         //Temporärer Fehler: #pdStatus = 80A7, 80B5, 80C0, 80C1, 80C2, 80C3 oder 80C4 zulassen und nocheinmal versuchen
         IF NOT (#pwWord1 = DW#16#80A7) AND NOT (#pwWord1 = DW#16#80B5) AND NOT (#pwWord1 = DW#16#80C0) AND
           NOT (#pwWord1 = DW#16#80C1) AND NOT (#pwWord1 = DW#16#80C2) AND NOT (#pwWord1 = DW#16#80C3) AND
           NOT (#pwWord1 = DW#16#80C4) THEN

           // Wiederholungsauftrag wieder zurücknehmen
           #sbWrStart2 := False;
           #sbRdStart2 := False;
           #sbWrite := False;

           // Fehler ausgeben 
           #sbError := #sbRdError;

         ELSE
           // Fehlerwiederholauftrag ??                   
           IF #siErrorCount = #siMaxErrCount THEN

             // Wiederholungsauftrag wieder zurücknehmen
             #sbWrStart2 := False;
             #sbRdStart2 := False;
             #sbWrite := False;

             //Fehlerzähler zurücksetzen
             #siErrorCount := 0;


             // Fehler ausgeben 
             #sbError := #sbRdError;

             // nix tun bis Zähler überläuft
           ELSE
             #siErrorCount := #siErrorCount + 1;
           END_IF;
         END_IF;

         // Fehler : die Auftragsreferenz der Antwort übertimmt nicht mit der Auftragsreferenz der Anfrage überein
       ELSIF NOT (#siReqRef = BYTE_TO_INT(#sxRespParaMulti.sxHeader.syReqRef)) AND NOT #sbRdBusy AND #pbValidSFB THEN
         #siErrorId := 1;
         #sbError := True;
         #sbDone := False;

         // Wiederholungsauftrag wieder zurücknehmen
         #sbWrStart2 := False;
         #sbRdStart2 := False;
         #sbWrite := False;

         // Fehler : falsche Auftragskennung zurück erhalten    
       ELSIF NOT (#sxRespParaMulti.sxHeader.syReqId = B#16#82 OR #sxRespParaMulti.sxHeader.syReqId = B#16#02) AND
         NOT #sbRdBusy AND #pbValidSFB THEN
         #siErrorId := 1;
         #sbError := True;
         #sbDone := False;

         // Wiederholungsauftrag wieder zurücknehmen
         #sbWrStart2 := False;
         #sbRdStart2 := False;
         #sbWrite := False;

         // Fehler : die angeforderte Anzahl Parameter entspricht nicht der übermittelten Anzahl Parameter überein
       ELSIF NOT (#sxRespParaMulti.sxHeader.syParaNo = B#16#01) AND NOT #sbRdBusy AND #pbValidSFB THEN
         #siErrorId := 1;
         #sbError := True;
         #sbDone := False;

         // Wiederholungsauftrag wieder zurücknehmen
         #sbWrStart2 := False;
         #sbRdStart2 := False;
         #sbWrite := False;

         // Fehler : die Achse entspricht nicht der übergebenen Achse
       ELSIF NOT (#syAxisNo = #sxRespParaMulti.sxHeader.syAxisNo) AND NOT #sbRdBusy AND #pbValidSFB THEN
         #siErrorId := 1;
         #sbError := True;
         #sbDone := False;

         // Wiederholungsauftrag wieder zurücknehmen
         #sbWrStart2 := False;
         #sbRdStart2 := False;
         #sbWrite := False;

         // kein Fehler beim LESEN AZYKLISCH und Auftrag fertig 
       ELSIF NOT #sbRdBusy AND #pbValidSFB THEN

         // 2. Teilauftrag "Parameter schreiben bzw. ändern" negative Rückmeldung erhalten 
         IF #sxRespParaMulti.sxHeader.syReqId = B#16#82 THEN

           // die angefragten Parameter auswerten und im Puffer abspeichern
           // Format des Parameters auswerten, bei Format = Error Fehler auswerten 
           IF (BYTE_TO_INT(#sxRespParaMulti.sxData[1]) = 68) THEN

             // Fehlerwert ermitteln und abspeichern 
             // Format = Word, zwei Bytes zu übermitteltem Parameterwert zusammenfassen
             #pwWordHigh := SHL(IN := BYTE_TO_WORD(#sxRespParaMulti.sxData[3]), N := 8);
             #pwWordLow := BYTE_TO_WORD(#sxRespParaMulti.sxData[4]);
             #pwWord1 := #pwWordHigh XOR #pwWordLow;

             #sbError := True;

             // ermittelte Fehlernummer im Puffer zurücksetzen
             #ErrorNo := W#16#00;

             #ErrorNo := #pwWord1;

             // Die Fehlerhaftigkeit des erkannten Parameter in der Fehlernummer eintragen   
             #swParaError := #swParaError OR W#16#01;

           ELSE

             // Die Fehlerhaftigkeit des erkannten Parameter in der Fehlernummer löschen   
             #swParaError := #swParaError AND W#16#FFFE;

             // ermittelte Fehlernummer im Puffer zurücksetzen
             #ErrorNo := W#16#00;
           END_IF;
         END_IF; // 2. Teilauftrag "Parameter schreiben bzw. ändern" negative Rückmeldung erhalten

         // Fehlerkennung zurücknehmen
         IF (#siErrorId = 3) OR (#siErrorId = 1) THEN
           #siErrorId := 0;
           #sbError := False;
         END_IF;

         #DiagId := W#16#00;

         // 2. Teilauftrag "Parameter schreiben bzw. ändern" ist abgeschlossen
         #sbRdStart2 := False;
         #sbWrite := False;

       END_IF; // kein Fehler beim LESEN AZYKLISCH und Auftrag fertig 
     END_IF; // vom 2. Teilauftrag "Parameter schreiben bzw. ändern" die Antwort abwarten und dann auswerten 
   END_IF; // Auftrag "Parameter schreiben" wurde ausgelöst

   #pdDWordHigh := SHL(IN := INT_TO_DWORD(#siErrorId), N := 16);
   #pdDWordLow := WORD_TO_DWORD(#swParaError);

   // ermittelter Parameterwert eintragen (Word)
   #ErrorId := #pdDWordHigh XOR #pdDWordLow;

   // Initialisierung von Ausgängen
   #Busy := #sbBusy;
   #Error := #sbError;
   #Format := #syFormat;
   // Änderung wegen verhalten von Ready  
   #Done := #sbDone;
   // Prüfen, ob Auftrag abgeschlossen ist
   IF ((#Error OR #Done) AND NOT #sbReady) THEN
     #Ready := True;
     #sbReady := True;
   ELSE
     #Ready := False;
   END_IF;
END_FUNCTION_BLOCK

FUNCTION_BLOCK "SevroStart&PosCheck"   // FB4073, LAD
{ S7_Optimized_Access := 'TRUE' }
// stored: AutoNumber false, MemoryReserve 100, SetENOAutomatically false
   VAR_INPUT
      iRef_Homed { ExternalAccessible := 'False'; ExternalVisible := 'False'; ExternalWritable := 'False'} : Bool;
      iStandstill { ExternalAccessible := 'False'; ExternalVisible := 'False'; ExternalWritable := 'False'} : Bool;
      iReset : Bool;
      interlcok : Bool;   // 启动互锁
      "iActual Posi" { ExternalAccessible := 'False'; ExternalVisible := 'False'; ExternalWritable := 'False'} : DInt;
      "iTol+" { ExternalAccessible := 'False'; ExternalVisible := 'False'; ExternalWritable := 'False'} : DInt;
      "iTol-" { ExternalAccessible := 'False'; ExternalVisible := 'False'; ExternalWritable := 'False'} : DInt;
      iStartTon : Time := T#200ms;   // 启动延迟
   END_VAR
   VAR_OUTPUT
      oStartPos : Bool;   // 启动
      DoublePosError : Bool;   // 多位置触发
   END_VAR
   VAR_IN_OUT
      ioPoint : Array[0..39] of Struct
         Start : Bool;
         Achieve : Bool;
      END_STRUCT;
      ioList : "PosList";
      ioPosNumberSelect : Int;   // 位置启动
   END_VAR
   VAR
      TON : Array[0..1] of TON_TIME;
      StartCount { S7_SetPoint := 'True'} : Int;   // 启动计数
   END_VAR
   VAR_TEMP
      "Actual Posi+Tol" : DInt;
      "Actual Posi-Tol" : DInt;
      Index : Array[0..7] of Int;   // 位置启动
      PosStart : Bool;
   END_VAR
   VAR_TEMP   // added for the SCL form of the ladder/FBD networks
      _w1 : Bool;
   END_VAR
BEGIN

REGION Network 1 (SCL): 检查当前启动位置号
   #Index[1] := 0;
   #PosStart := false;
   FOR #Index[1] := 0 TO 39 DO
       IF #ioPoint[#Index[1]].Start THEN

           #ioPosNumberSelect := #Index[1];//当前启动位置号
           #PosStart := TRUE;
           EXIT;
       END_IF;
   END_FOR;
   #Index[2] := 0;
   #StartCount := 0;
   FOR #Index[2] := 0 TO 39 DO
       IF #ioPoint[#Index[2]].Start THEN

           #StartCount := #StartCount+1;//当前启动位置号


       END_IF;
       IF #Index[2] = 39 THEN

           EXIT;
       END_IF;

   END_FOR;
END_REGION

REGION Network 2: 位置给定
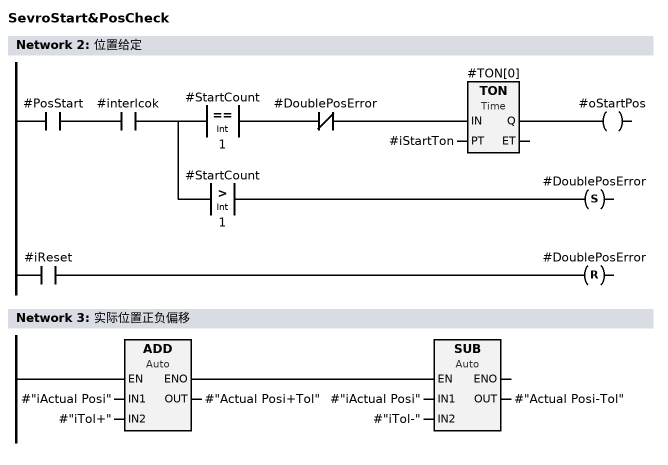
   RUNG wire#powerrail
      Contact( #PosStart )
      Contact( #interlcok )
      wire#w1
      { S7_Templates := "SrcType := Int" } EQ_Contact(in1 := #StartCount, in2 := 1)
      I_Contact( #DoublePosError )
      { S7_Templates := "time_type := Time" } #TON[0].TON(pt := #iStartTon, et =>)
      Coil( #oStartPos )
   END_RUNG
   RUNG wire#w1
      { S7_Templates := "SrcType := Int" } GT_Contact(in1 := #StartCount, in2 := 1)
      S_Coil( #DoublePosError )
   END_RUNG
   RUNG wire#powerrail
      Contact( #iReset )
      R_Coil( #DoublePosError )
   END_RUNG
   // the same network as SCL:
   #_w1 := #PosStart AND #interlcok;
   #TON[0].TON(IN := #_w1 AND (#StartCount = 1) AND NOT #DoublePosError, PT := #iStartTon);
   #oStartPos := #TON[0].Q;
   IF #_w1 AND (#StartCount > 1) THEN #DoublePosError := TRUE; END_IF;
   IF #iReset THEN #DoublePosError := FALSE; END_IF;
END_REGION

REGION Network 3: 实际位置正负偏移
   RUNG wire#powerrail
      Add(in1 := #"iActual Posi", in2 := #"iTol+", out => #"Actual Posi+Tol")
      Sub(in1 := #"iActual Posi", in2 := #"iTol-", out => #"Actual Posi-Tol")
   END_RUNG
   // the same network as SCL:
   #"Actual Posi+Tol" := #"iActual Posi" + #"iTol+";
   #"Actual Posi-Tol" := #"iActual Posi" - #"iTol-";
END_REGION

REGION Network 4 (SCL): 位置检查


   #Index[3] := 0;
   FOR #Index[3] := 0 TO 39 DO
       IF #ioList.List[ #Index[3]].Pos>= #"Actual Posi-Tol"
           AND #ioList.List[ #Index[3]].Pos<= #"Actual Posi+Tol"
       THEN
         #ioPoint[#Index[3]].Achieve := TRUE;
       ELSE
           #ioPoint[#Index[3]].Achieve := FALSE;
       END_IF;
   END_FOR;
END_REGION
END_FUNCTION_BLOCK

FUNCTION "Motorr" : Void   // FC3100, LAD
{ S7_Optimized_Access := 'TRUE' }
// stored: AutoNumber false, SetENOAutomatically false
   VAR_TEMP   // added for the SCL form of the ladder/FBD networks
      _w1 : Bool;
      _w2 : Bool;
   END_VAR
BEGIN

REGION Network 1: H-shaftLifting_Motor
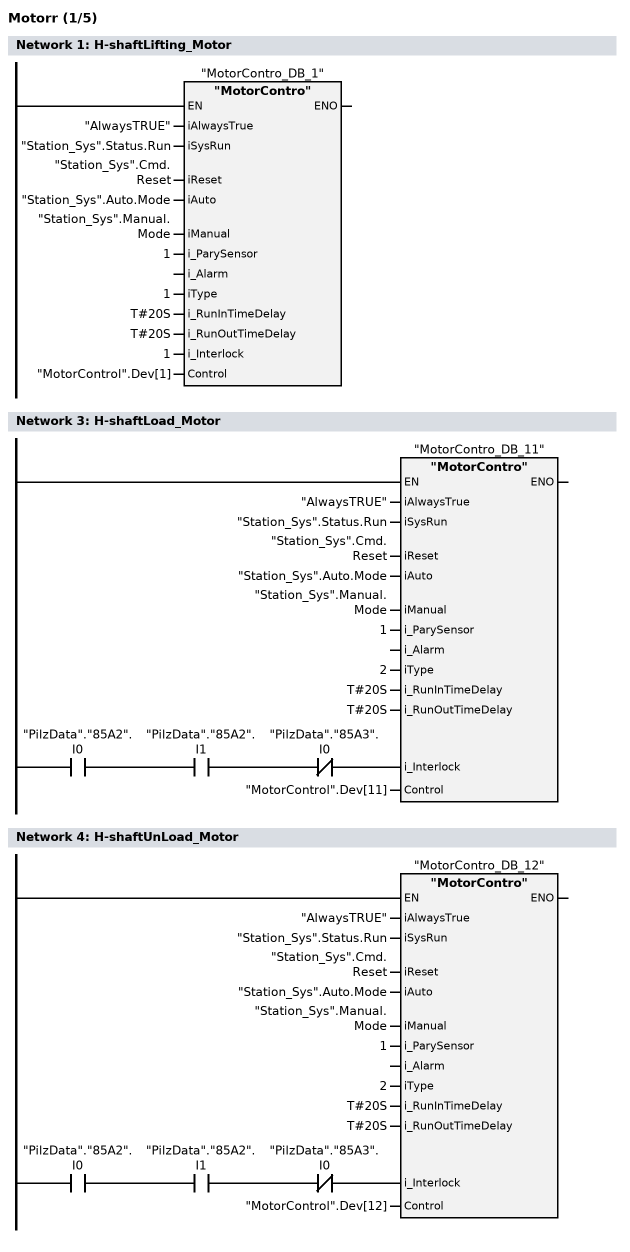
   RUNG wire#powerrail
      "MotorContro_DB_1"(iAlwaysTrue := "AlwaysTRUE", iSysRun := "Station_Sys".Status.Run, iReset := "Station_Sys".Cmd.Reset, iAuto := "Station_Sys".Auto.Mode, iManual := "Station_Sys".Manual.Mode, i_ParySensor := 1, i_Alarm :=, iType := 1, i_RunInTimeDelay := T#20S, i_RunOutTimeDelay := T#20S, i_Interlock := 1, Control := "MotorControl".Dev[1])
   END_RUNG
   // the same network as SCL:
   "MotorContro_DB_1"(iAlwaysTrue := "AlwaysTRUE",   // "MotorContro"
                      iSysRun := "Station_Sys".Status.Run,
                      iReset := "Station_Sys".Cmd.Reset,
                      iAuto := "Station_Sys".Auto.Mode,
                      iManual := "Station_Sys".Manual.Mode,
                      i_ParySensor := 1,
                      iType := 1,
                      i_RunInTimeDelay := T#20S,
                      i_RunOutTimeDelay := T#20S,
                      i_Interlock := 1,
                      Control := "MotorControl".Dev[1]);
END_REGION

REGION Network 2 (SCL): H-shaftLifting_Motor_OutPut
   "oH-shaftLifting_Start" := "MotorControl".Dev[1].OutControl.o_Start;
   "oH-shaftLifting_CCWStart" := "MotorControl".Dev[1].OutControl.o_CCWStart ;
   "oH-shaftLifting_SpeedChange" := "MotorControl".Dev[1].OutControl.o_SpeedChanged;
END_REGION

REGION Network 3: H-shaftLoad_Motor
   RUNG wire#powerrail
      "MotorContro_DB_11"(i_Interlock := wire#w1, iAlwaysTrue := "AlwaysTRUE", iSysRun := "Station_Sys".Status.Run, iReset := "Station_Sys".Cmd.Reset, iAuto := "Station_Sys".Auto.Mode, iManual := "Station_Sys".Manual.Mode, i_ParySensor := 1, i_Alarm :=, iType := 2, i_RunInTimeDelay := T#20S, i_RunOutTimeDelay := T#20S, Control := "MotorControl".Dev[11])
   END_RUNG
   RUNG wire#powerrail
      Contact( "PilzData"."85A2".I0 )
      Contact( "PilzData"."85A2".I1 )
      I_Contact( "PilzData"."85A3".I0 )
   END_RUNG wire#w1
   // the same network as SCL:
   "MotorContro_DB_11"(iAlwaysTrue := "AlwaysTRUE",   // "MotorContro"
                       iSysRun := "Station_Sys".Status.Run,
                       iReset := "Station_Sys".Cmd.Reset,
                       iAuto := "Station_Sys".Auto.Mode,
                       iManual := "Station_Sys".Manual.Mode,
                       i_ParySensor := 1,
                       iType := 2,
                       i_RunInTimeDelay := T#20S,
                       i_RunOutTimeDelay := T#20S,
                       i_Interlock := "PilzData"."85A2".I0 AND "PilzData"."85A2".I1 AND NOT "PilzData"."85A3".I0,
                       Control := "MotorControl".Dev[11]);
END_REGION

REGION Network 4: H-shaftUnLoad_Motor
   RUNG wire#powerrail
      "MotorContro_DB_12"(i_Interlock := wire#w1, iAlwaysTrue := "AlwaysTRUE", iSysRun := "Station_Sys".Status.Run, iReset := "Station_Sys".Cmd.Reset, iAuto := "Station_Sys".Auto.Mode, iManual := "Station_Sys".Manual.Mode, i_ParySensor := 1, i_Alarm :=, iType := 2, i_RunInTimeDelay := T#20S, i_RunOutTimeDelay := T#20S, Control := "MotorControl".Dev[12])
   END_RUNG
   RUNG wire#powerrail
      Contact( "PilzData"."85A2".I0 )
      Contact( "PilzData"."85A2".I1 )
      I_Contact( "PilzData"."85A3".I0 )
   END_RUNG wire#w1
   // the same network as SCL:
   "MotorContro_DB_12"(iAlwaysTrue := "AlwaysTRUE",   // "MotorContro"
                       iSysRun := "Station_Sys".Status.Run,
                       iReset := "Station_Sys".Cmd.Reset,
                       iAuto := "Station_Sys".Auto.Mode,
                       iManual := "Station_Sys".Manual.Mode,
                       i_ParySensor := 1,
                       iType := 2,
                       i_RunInTimeDelay := T#20S,
                       i_RunOutTimeDelay := T#20S,
                       i_Interlock := "PilzData"."85A2".I0 AND "PilzData"."85A2".I1 AND NOT "PilzData"."85A3".I0,
                       Control := "MotorControl".Dev[12]);
END_REGION

REGION Network 5 (SCL): H-shaftLifting_Motor_OutPut / H-shaftLoad_Motor_OutPut
   "oH-shaftLoading_CW" := "MotorControl".Dev[11].OutControl.o_Start;
   "oH-shaftLoading_CCW" := "MotorControl".Dev[11].OutControl.o_CCWStart OR ("Station_Sys".Auto.Mode AND "AutoProcessControl".Global.H.EmptyPallet);

   "oH-shaftTake_CW" := "MotorControl".Dev[12].OutControl.o_Start;
END_REGION

REGION Network 6: Auto MotorStop
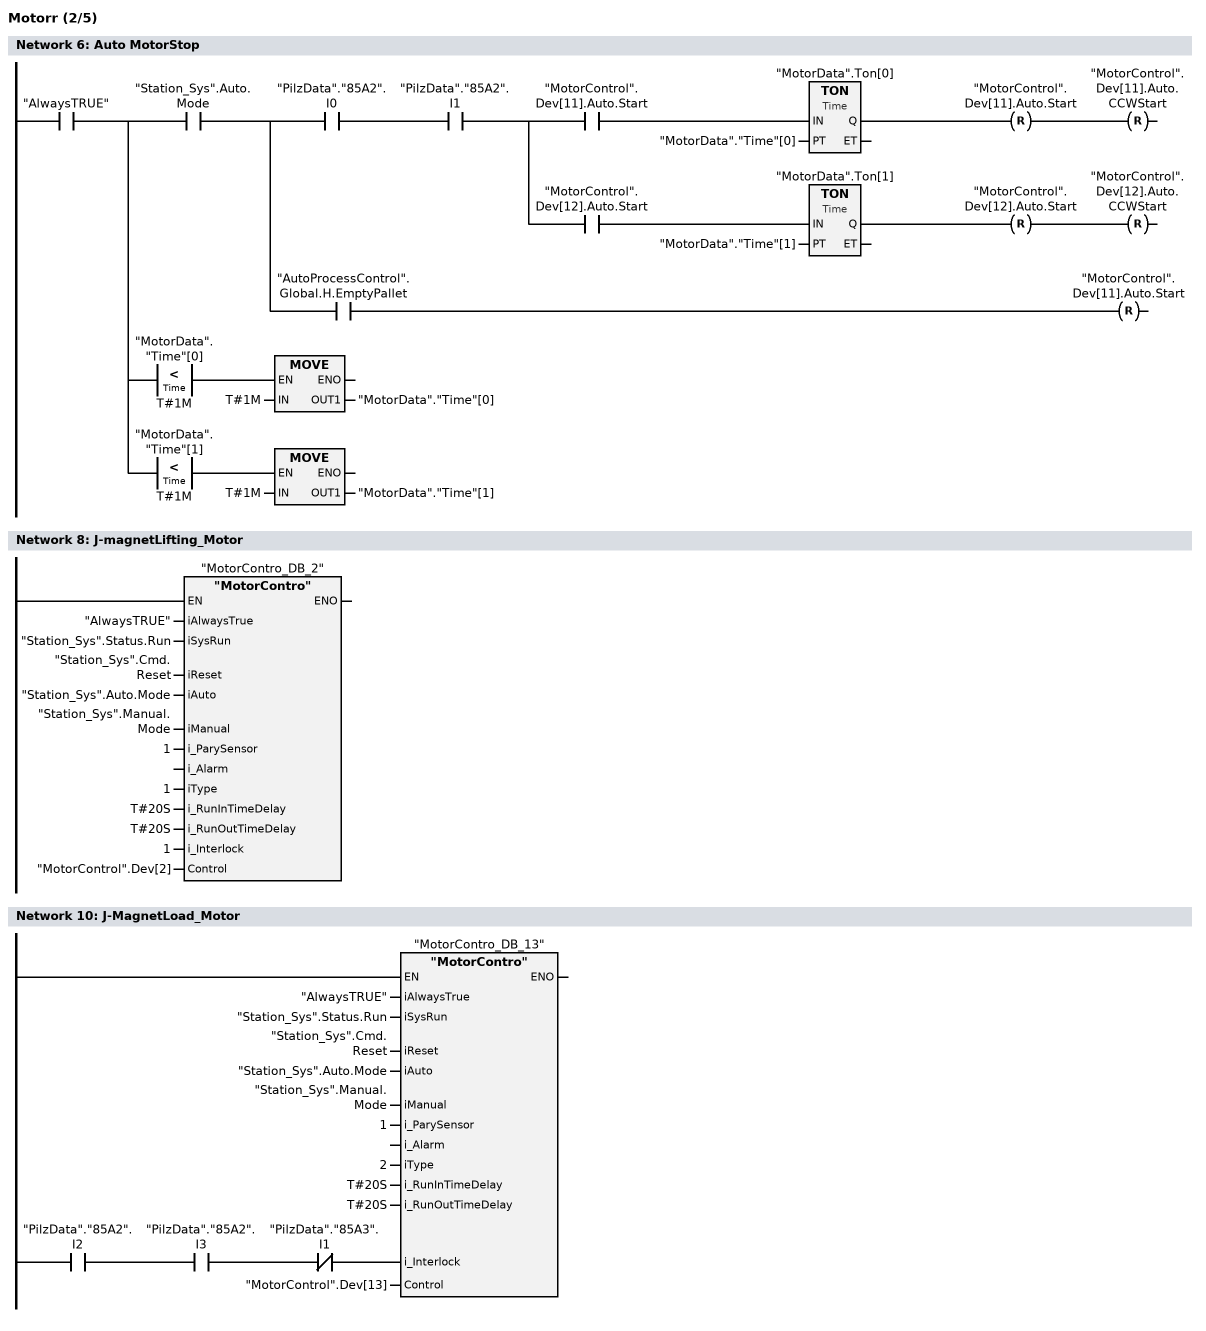
   RUNG wire#powerrail
      Contact( "AlwaysTRUE" )
      wire#w1
      Contact( "Station_Sys".Auto.Mode )
      wire#w2
      Contact( "PilzData"."85A2".I0 )
      Contact( "PilzData"."85A2".I1 )
      wire#w3
      Contact( "MotorControl".Dev[11].Auto.Start )
      { S7_Templates := "time_type := Time" } "MotorData".Ton[0].TON(pt := "MotorData"."Time"[0], et =>)
      R_Coil( "MotorControl".Dev[11].Auto.Start )
      R_Coil( "MotorControl".Dev[11].Auto.CCWStart )
   END_RUNG
   RUNG wire#w3
      Contact( "MotorControl".Dev[12].Auto.Start )
      { S7_Templates := "time_type := Time" } "MotorData".Ton[1].TON(pt := "MotorData"."Time"[1], et =>)
      R_Coil( "MotorControl".Dev[12].Auto.Start )
      R_Coil( "MotorControl".Dev[12].Auto.CCWStart )
   END_RUNG
   RUNG wire#w2
      Contact( "AutoProcessControl".Global.H.EmptyPallet )
      R_Coil( "MotorControl".Dev[11].Auto.Start )
   END_RUNG
   RUNG wire#w1
      { S7_Templates := "SrcType := Time" } LT_Contact(in1 := "MotorData"."Time"[0], in2 := T#1M)
      Move(in := T#1M, out1 => "MotorData"."Time"[0])
   END_RUNG
   RUNG wire#w1
      { S7_Templates := "SrcType := Time" } LT_Contact(in1 := "MotorData"."Time"[1], in2 := T#1M)
      Move(in := T#1M, out1 => "MotorData"."Time"[1])
   END_RUNG
   // the same network as SCL:
   #_w1 := "AlwaysTRUE" AND "Station_Sys".Auto.Mode;
   #_w2 := #_w1 AND "PilzData"."85A2".I0 AND "PilzData"."85A2".I1;
   "MotorData".Ton[0].TON(IN := #_w2 AND "MotorControl".Dev[11].Auto.Start, PT := "MotorData"."Time"[0]);
   IF "MotorData".Ton[0].Q THEN
       "MotorControl".Dev[11].Auto.Start := FALSE;
       "MotorControl".Dev[11].Auto.CCWStart := FALSE;
   END_IF;
   "MotorData".Ton[1].TON(IN := #_w2 AND "MotorControl".Dev[12].Auto.Start, PT := "MotorData"."Time"[1]);
   IF "MotorData".Ton[1].Q THEN
       "MotorControl".Dev[12].Auto.Start := FALSE;
       "MotorControl".Dev[12].Auto.CCWStart := FALSE;
   END_IF;
   IF #_w1 AND "AutoProcessControl".Global.H.EmptyPallet THEN
       "MotorControl".Dev[11].Auto.Start := FALSE;
   END_IF;
   IF "AlwaysTRUE" AND ("MotorData"."Time"[0] < T#1M) THEN "MotorData"."Time"[0] := T#1M; END_IF;
   IF "AlwaysTRUE" AND ("MotorData"."Time"[1] < T#1M) THEN "MotorData"."Time"[1] := T#1M; END_IF;
END_REGION

REGION Network 8: J-magnetLifting_Motor
   RUNG wire#powerrail
      "MotorContro_DB_2"(iAlwaysTrue := "AlwaysTRUE", iSysRun := "Station_Sys".Status.Run, iReset := "Station_Sys".Cmd.Reset, iAuto := "Station_Sys".Auto.Mode, iManual := "Station_Sys".Manual.Mode, i_ParySensor := 1, i_Alarm :=, iType := 1, i_RunInTimeDelay := T#20S, i_RunOutTimeDelay := T#20S, i_Interlock := 1, Control := "MotorControl".Dev[2])
   END_RUNG
   // the same network as SCL:
   "MotorContro_DB_2"(iAlwaysTrue := "AlwaysTRUE",   // "MotorContro"
                      iSysRun := "Station_Sys".Status.Run,
                      iReset := "Station_Sys".Cmd.Reset,
                      iAuto := "Station_Sys".Auto.Mode,
                      iManual := "Station_Sys".Manual.Mode,
                      i_ParySensor := 1,
                      iType := 1,
                      i_RunInTimeDelay := T#20S,
                      i_RunOutTimeDelay := T#20S,
                      i_Interlock := 1,
                      Control := "MotorControl".Dev[2]);
END_REGION

REGION Network 9 (SCL): J-magnetLifting_Motor_OutPut
   "oJ-magnetLifting_Start" := "MotorControl".Dev[2].OutControl.o_Start;
   "oJ-magnetLifting_CCWStart" := "MotorControl".Dev[2].OutControl.o_CCWStart;
   "oJ-magnetLifting_SpeedChange" := "MotorControl".Dev[2].OutControl.o_SpeedChanged;
END_REGION

REGION Network 10: J-MagnetLoad_Motor
   RUNG wire#powerrail
      "MotorContro_DB_13"(i_Interlock := wire#w1, iAlwaysTrue := "AlwaysTRUE", iSysRun := "Station_Sys".Status.Run, iReset := "Station_Sys".Cmd.Reset, iAuto := "Station_Sys".Auto.Mode, iManual := "Station_Sys".Manual.Mode, i_ParySensor := 1, i_Alarm :=, iType := 2, i_RunInTimeDelay := T#20S, i_RunOutTimeDelay := T#20S, Control := "MotorControl".Dev[13])
   END_RUNG
   RUNG wire#powerrail
      Contact( "PilzData"."85A2".I2 )
      Contact( "PilzData"."85A2".I3 )
      I_Contact( "PilzData"."85A3".I1 )
   END_RUNG wire#w1
   // the same network as SCL:
   "MotorContro_DB_13"(iAlwaysTrue := "AlwaysTRUE",   // "MotorContro"
                       iSysRun := "Station_Sys".Status.Run,
                       iReset := "Station_Sys".Cmd.Reset,
                       iAuto := "Station_Sys".Auto.Mode,
                       iManual := "Station_Sys".Manual.Mode,
                       i_ParySensor := 1,
                       iType := 2,
                       i_RunInTimeDelay := T#20S,
                       i_RunOutTimeDelay := T#20S,
                       i_Interlock := "PilzData"."85A2".I2 AND "PilzData"."85A2".I3 AND NOT "PilzData"."85A3".I1,
                       Control := "MotorControl".Dev[13]);
END_REGION

REGION Network 11: J-MagnetUnLoad_Motor
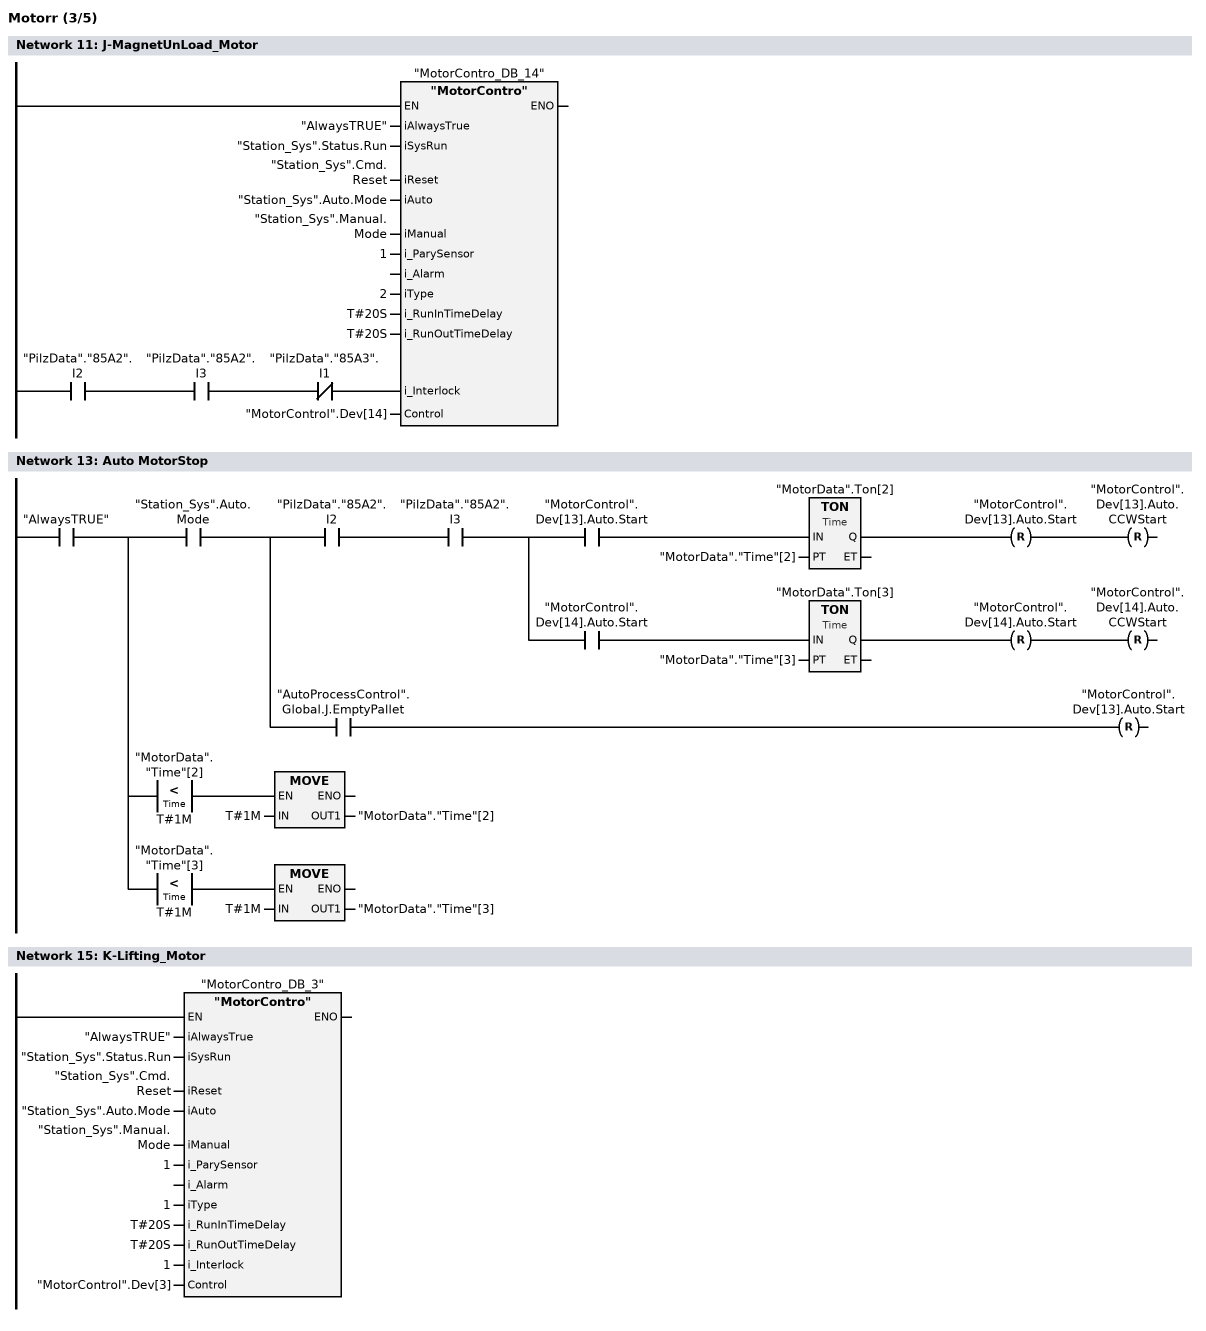
   RUNG wire#powerrail
      "MotorContro_DB_14"(i_Interlock := wire#w1, iAlwaysTrue := "AlwaysTRUE", iSysRun := "Station_Sys".Status.Run, iReset := "Station_Sys".Cmd.Reset, iAuto := "Station_Sys".Auto.Mode, iManual := "Station_Sys".Manual.Mode, i_ParySensor := 1, i_Alarm :=, iType := 2, i_RunInTimeDelay := T#20S, i_RunOutTimeDelay := T#20S, Control := "MotorControl".Dev[14])
   END_RUNG
   RUNG wire#powerrail
      Contact( "PilzData"."85A2".I2 )
      Contact( "PilzData"."85A2".I3 )
      I_Contact( "PilzData"."85A3".I1 )
   END_RUNG wire#w1
   // the same network as SCL:
   "MotorContro_DB_14"(iAlwaysTrue := "AlwaysTRUE",   // "MotorContro"
                       iSysRun := "Station_Sys".Status.Run,
                       iReset := "Station_Sys".Cmd.Reset,
                       iAuto := "Station_Sys".Auto.Mode,
                       iManual := "Station_Sys".Manual.Mode,
                       i_ParySensor := 1,
                       iType := 2,
                       i_RunInTimeDelay := T#20S,
                       i_RunOutTimeDelay := T#20S,
                       i_Interlock := "PilzData"."85A2".I2 AND "PilzData"."85A2".I3 AND NOT "PilzData"."85A3".I1,
                       Control := "MotorControl".Dev[14]);
END_REGION

REGION Network 12 (SCL): H-shaftLifting_Motor_OutPut / J-Magnet_Motor_OutPut
   "J-magnet Loading _CW" := "MotorControl".Dev[13].OutControl.o_Start;
   "J-magnet Loading _CCW" := "MotorControl".Dev[13].OutControl.o_CCWStart OR ("Station_Sys".Auto.Mode AND "AutoProcessControl".Global.J.EmptyPallet);

   "J-magnet Take _CW" := "MotorControl".Dev[14].OutControl.o_Start;
END_REGION

REGION Network 13: Auto MotorStop
   RUNG wire#powerrail
      Contact( "AlwaysTRUE" )
      wire#w1
      Contact( "Station_Sys".Auto.Mode )
      wire#w2
      Contact( "PilzData"."85A2".I2 )
      Contact( "PilzData"."85A2".I3 )
      wire#w3
      Contact( "MotorControl".Dev[13].Auto.Start )
      { S7_Templates := "time_type := Time" } "MotorData".Ton[2].TON(pt := "MotorData"."Time"[2], et =>)
      R_Coil( "MotorControl".Dev[13].Auto.Start )
      R_Coil( "MotorControl".Dev[13].Auto.CCWStart )
   END_RUNG
   RUNG wire#w3
      Contact( "MotorControl".Dev[14].Auto.Start )
      { S7_Templates := "time_type := Time" } "MotorData".Ton[3].TON(pt := "MotorData"."Time"[3], et =>)
      R_Coil( "MotorControl".Dev[14].Auto.Start )
      R_Coil( "MotorControl".Dev[14].Auto.CCWStart )
   END_RUNG
   RUNG wire#w2
      Contact( "AutoProcessControl".Global.J.EmptyPallet )
      R_Coil( "MotorControl".Dev[13].Auto.Start )
   END_RUNG
   RUNG wire#w1
      { S7_Templates := "SrcType := Time" } LT_Contact(in1 := "MotorData"."Time"[2], in2 := T#1M)
      Move(in := T#1M, out1 => "MotorData"."Time"[2])
   END_RUNG
   RUNG wire#w1
      { S7_Templates := "SrcType := Time" } LT_Contact(in1 := "MotorData"."Time"[3], in2 := T#1M)
      Move(in := T#1M, out1 => "MotorData"."Time"[3])
   END_RUNG
   // the same network as SCL:
   #_w1 := "AlwaysTRUE" AND "Station_Sys".Auto.Mode;
   #_w2 := #_w1 AND "PilzData"."85A2".I2 AND "PilzData"."85A2".I3;
   "MotorData".Ton[2].TON(IN := #_w2 AND "MotorControl".Dev[13].Auto.Start, PT := "MotorData"."Time"[2]);
   IF "MotorData".Ton[2].Q THEN
       "MotorControl".Dev[13].Auto.Start := FALSE;
       "MotorControl".Dev[13].Auto.CCWStart := FALSE;
   END_IF;
   "MotorData".Ton[3].TON(IN := #_w2 AND "MotorControl".Dev[14].Auto.Start, PT := "MotorData"."Time"[3]);
   IF "MotorData".Ton[3].Q THEN
       "MotorControl".Dev[14].Auto.Start := FALSE;
       "MotorControl".Dev[14].Auto.CCWStart := FALSE;
   END_IF;
   IF #_w1 AND "AutoProcessControl".Global.J.EmptyPallet THEN
       "MotorControl".Dev[13].Auto.Start := FALSE;
   END_IF;
   IF "AlwaysTRUE" AND ("MotorData"."Time"[2] < T#1M) THEN "MotorData"."Time"[2] := T#1M; END_IF;
   IF "AlwaysTRUE" AND ("MotorData"."Time"[3] < T#1M) THEN "MotorData"."Time"[3] := T#1M; END_IF;
END_REGION

REGION Network 15: K-Lifting_Motor
   RUNG wire#powerrail
      "MotorContro_DB_3"(iAlwaysTrue := "AlwaysTRUE", iSysRun := "Station_Sys".Status.Run, iReset := "Station_Sys".Cmd.Reset, iAuto := "Station_Sys".Auto.Mode, iManual := "Station_Sys".Manual.Mode, i_ParySensor := 1, i_Alarm :=, iType := 1, i_RunInTimeDelay := T#20S, i_RunOutTimeDelay := T#20S, i_Interlock := 1, Control := "MotorControl".Dev[3])
   END_RUNG
   // the same network as SCL:
   "MotorContro_DB_3"(iAlwaysTrue := "AlwaysTRUE",   // "MotorContro"
                      iSysRun := "Station_Sys".Status.Run,
                      iReset := "Station_Sys".Cmd.Reset,
                      iAuto := "Station_Sys".Auto.Mode,
                      iManual := "Station_Sys".Manual.Mode,
                      i_ParySensor := 1,
                      iType := 1,
                      i_RunInTimeDelay := T#20S,
                      i_RunOutTimeDelay := T#20S,
                      i_Interlock := 1,
                      Control := "MotorControl".Dev[3]);
END_REGION

REGION Network 16 (SCL): K-Lifting_Motor_OutPut
   "oK-Lifting3_Start" := "MotorControl".Dev[3].OutControl.o_Start;
   "oK-Lifting3_CCWStart" := "MotorControl".Dev[3].OutControl.o_CCWStart;
   "oK-Lifting3_SpeedChange" := "MotorControl".Dev[3].OutControl.o_SpeedChanged;
END_REGION

REGION Network 17: K-ReserveLoad_Motor
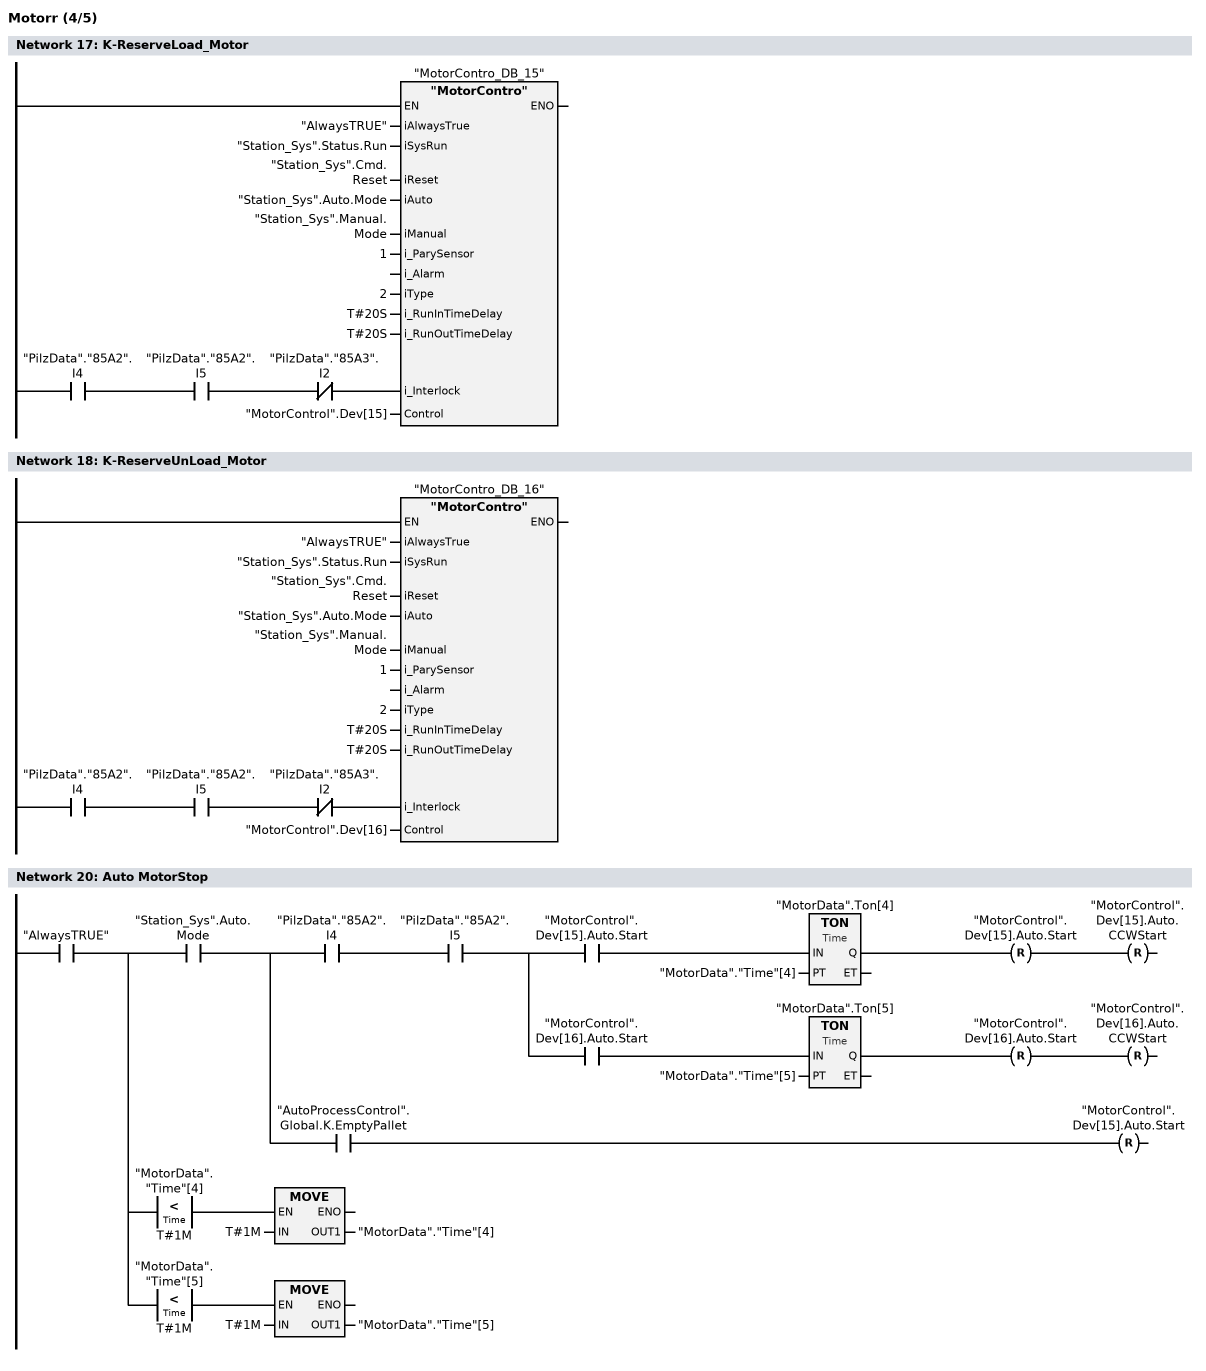
   RUNG wire#powerrail
      "MotorContro_DB_15"(i_Interlock := wire#w1, iAlwaysTrue := "AlwaysTRUE", iSysRun := "Station_Sys".Status.Run, iReset := "Station_Sys".Cmd.Reset, iAuto := "Station_Sys".Auto.Mode, iManual := "Station_Sys".Manual.Mode, i_ParySensor := 1, i_Alarm :=, iType := 2, i_RunInTimeDelay := T#20S, i_RunOutTimeDelay := T#20S, Control := "MotorControl".Dev[15])
   END_RUNG
   RUNG wire#powerrail
      Contact( "PilzData"."85A2".I4 )
      Contact( "PilzData"."85A2".I5 )
      I_Contact( "PilzData"."85A3".I2 )
   END_RUNG wire#w1
   // the same network as SCL:
   "MotorContro_DB_15"(iAlwaysTrue := "AlwaysTRUE",   // "MotorContro"
                       iSysRun := "Station_Sys".Status.Run,
                       iReset := "Station_Sys".Cmd.Reset,
                       iAuto := "Station_Sys".Auto.Mode,
                       iManual := "Station_Sys".Manual.Mode,
                       i_ParySensor := 1,
                       iType := 2,
                       i_RunInTimeDelay := T#20S,
                       i_RunOutTimeDelay := T#20S,
                       i_Interlock := "PilzData"."85A2".I4 AND "PilzData"."85A2".I5 AND NOT "PilzData"."85A3".I2,
                       Control := "MotorControl".Dev[15]);
END_REGION

REGION Network 18: K-ReserveUnLoad_Motor
   RUNG wire#powerrail
      "MotorContro_DB_16"(i_Interlock := wire#w1, iAlwaysTrue := "AlwaysTRUE", iSysRun := "Station_Sys".Status.Run, iReset := "Station_Sys".Cmd.Reset, iAuto := "Station_Sys".Auto.Mode, iManual := "Station_Sys".Manual.Mode, i_ParySensor := 1, i_Alarm :=, iType := 2, i_RunInTimeDelay := T#20S, i_RunOutTimeDelay := T#20S, Control := "MotorControl".Dev[16])
   END_RUNG
   RUNG wire#powerrail
      Contact( "PilzData"."85A2".I4 )
      Contact( "PilzData"."85A2".I5 )
      I_Contact( "PilzData"."85A3".I2 )
   END_RUNG wire#w1
   // the same network as SCL:
   "MotorContro_DB_16"(iAlwaysTrue := "AlwaysTRUE",   // "MotorContro"
                       iSysRun := "Station_Sys".Status.Run,
                       iReset := "Station_Sys".Cmd.Reset,
                       iAuto := "Station_Sys".Auto.Mode,
                       iManual := "Station_Sys".Manual.Mode,
                       i_ParySensor := 1,
                       iType := 2,
                       i_RunInTimeDelay := T#20S,
                       i_RunOutTimeDelay := T#20S,
                       i_Interlock := "PilzData"."85A2".I4 AND "PilzData"."85A2".I5 AND NOT "PilzData"."85A3".I2,
                       Control := "MotorControl".Dev[16]);
END_REGION

REGION Network 19 (SCL): H-shaftLifting_Motor_OutPut / K-Reserve_Motor_OutPut
   "K-Loading _CW" := "MotorControl".Dev[15].OutControl.o_Start;
   "K-Loading _CCW" := "MotorControl".Dev[15].OutControl.o_CCWStart OR ("Station_Sys".Auto.Mode AND "AutoProcessControl".Global.K.EmptyPallet);

   "K-Take _CW" := "MotorControl".Dev[16].OutControl.o_Start;
END_REGION

REGION Network 20: Auto MotorStop
   RUNG wire#powerrail
      Contact( "AlwaysTRUE" )
      wire#w1
      Contact( "Station_Sys".Auto.Mode )
      wire#w2
      Contact( "PilzData"."85A2".I4 )
      Contact( "PilzData"."85A2".I5 )
      wire#w3
      Contact( "MotorControl".Dev[15].Auto.Start )
      { S7_Templates := "time_type := Time" } "MotorData".Ton[4].TON(pt := "MotorData"."Time"[4], et =>)
      R_Coil( "MotorControl".Dev[15].Auto.Start )
      R_Coil( "MotorControl".Dev[15].Auto.CCWStart )
   END_RUNG
   RUNG wire#w3
      Contact( "MotorControl".Dev[16].Auto.Start )
      { S7_Templates := "time_type := Time" } "MotorData".Ton[5].TON(pt := "MotorData"."Time"[5], et =>)
      R_Coil( "MotorControl".Dev[16].Auto.Start )
      R_Coil( "MotorControl".Dev[16].Auto.CCWStart )
   END_RUNG
   RUNG wire#w2
      Contact( "AutoProcessControl".Global.K.EmptyPallet )
      R_Coil( "MotorControl".Dev[15].Auto.Start )
   END_RUNG
   RUNG wire#w1
      { S7_Templates := "SrcType := Time" } LT_Contact(in1 := "MotorData"."Time"[4], in2 := T#1M)
      Move(in := T#1M, out1 => "MotorData"."Time"[4])
   END_RUNG
   RUNG wire#w1
      { S7_Templates := "SrcType := Time" } LT_Contact(in1 := "MotorData"."Time"[5], in2 := T#1M)
      Move(in := T#1M, out1 => "MotorData"."Time"[5])
   END_RUNG
   // the same network as SCL:
   #_w1 := "AlwaysTRUE" AND "Station_Sys".Auto.Mode;
   #_w2 := #_w1 AND "PilzData"."85A2".I4 AND "PilzData"."85A2".I5;
   "MotorData".Ton[4].TON(IN := #_w2 AND "MotorControl".Dev[15].Auto.Start, PT := "MotorData"."Time"[4]);
   IF "MotorData".Ton[4].Q THEN
       "MotorControl".Dev[15].Auto.Start := FALSE;
       "MotorControl".Dev[15].Auto.CCWStart := FALSE;
   END_IF;
   "MotorData".Ton[5].TON(IN := #_w2 AND "MotorControl".Dev[16].Auto.Start, PT := "MotorData"."Time"[5]);
   IF "MotorData".Ton[5].Q THEN
       "MotorControl".Dev[16].Auto.Start := FALSE;
       "MotorControl".Dev[16].Auto.CCWStart := FALSE;
   END_IF;
   IF #_w1 AND "AutoProcessControl".Global.K.EmptyPallet THEN
       "MotorControl".Dev[15].Auto.Start := FALSE;
   END_IF;
   IF "AlwaysTRUE" AND ("MotorData"."Time"[4] < T#1M) THEN "MotorData"."Time"[4] := T#1M; END_IF;
   IF "AlwaysTRUE" AND ("MotorData"."Time"[5] < T#1M) THEN "MotorData"."Time"[5] := T#1M; END_IF;
END_REGION

REGION Network 22: L-Unloading_Motor
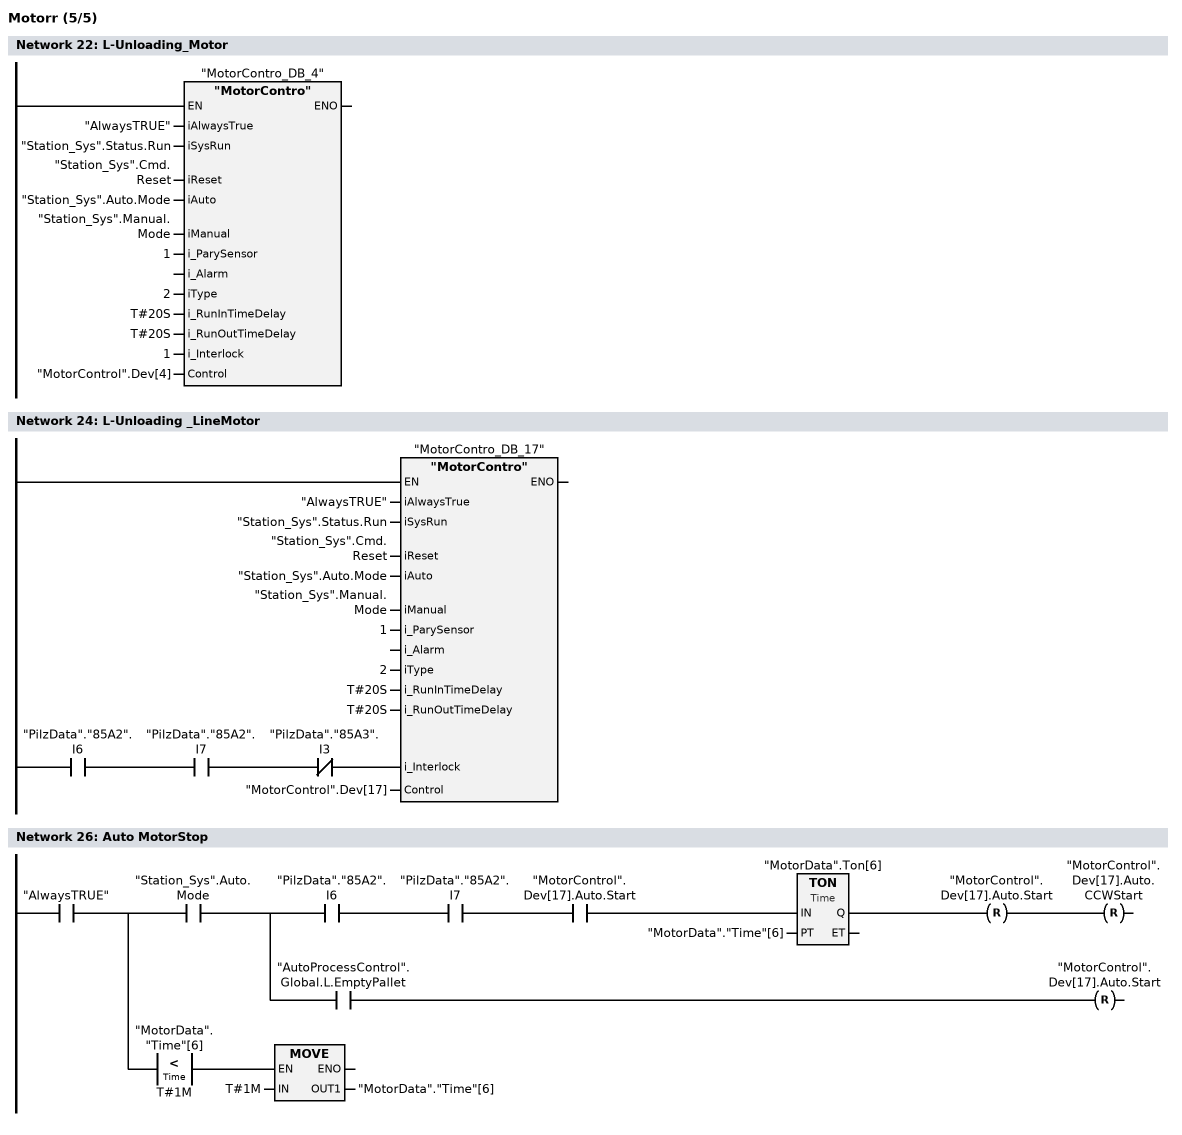
   RUNG wire#powerrail
      "MotorContro_DB_4"(iAlwaysTrue := "AlwaysTRUE", iSysRun := "Station_Sys".Status.Run, iReset := "Station_Sys".Cmd.Reset, iAuto := "Station_Sys".Auto.Mode, iManual := "Station_Sys".Manual.Mode, i_ParySensor := 1, i_Alarm :=, iType := 2, i_RunInTimeDelay := T#20S, i_RunOutTimeDelay := T#20S, i_Interlock := 1, Control := "MotorControl".Dev[4])
   END_RUNG
   // the same network as SCL:
   "MotorContro_DB_4"(iAlwaysTrue := "AlwaysTRUE",   // "MotorContro"
                      iSysRun := "Station_Sys".Status.Run,
                      iReset := "Station_Sys".Cmd.Reset,
                      iAuto := "Station_Sys".Auto.Mode,
                      iManual := "Station_Sys".Manual.Mode,
                      i_ParySensor := 1,
                      iType := 2,
                      i_RunInTimeDelay := T#20S,
                      i_RunOutTimeDelay := T#20S,
                      i_Interlock := 1,
                      Control := "MotorControl".Dev[4]);
END_REGION

REGION Network 23 (SCL): L-Unloading_Motor_OutPut
   "oL-Unloading_CW" := "MotorControl".Dev[4].OutControl.o_Start;
   "oL-Unloading_CCW" := "MotorControl".Dev[4].OutControl.o_CCWStart;
END_REGION

REGION Network 24: L-Unloading _LineMotor
   RUNG wire#powerrail
      "MotorContro_DB_17"(i_Interlock := wire#w1, iAlwaysTrue := "AlwaysTRUE", iSysRun := "Station_Sys".Status.Run, iReset := "Station_Sys".Cmd.Reset, iAuto := "Station_Sys".Auto.Mode, iManual := "Station_Sys".Manual.Mode, i_ParySensor := 1, i_Alarm :=, iType := 2, i_RunInTimeDelay := T#20S, i_RunOutTimeDelay := T#20S, Control := "MotorControl".Dev[17])
   END_RUNG
   RUNG wire#powerrail
      Contact( "PilzData"."85A2".I6 )
      Contact( "PilzData"."85A2".I7 )
      I_Contact( "PilzData"."85A3".I3 )
   END_RUNG wire#w1
   // the same network as SCL:
   "MotorContro_DB_17"(iAlwaysTrue := "AlwaysTRUE",   // "MotorContro"
                       iSysRun := "Station_Sys".Status.Run,
                       iReset := "Station_Sys".Cmd.Reset,
                       iAuto := "Station_Sys".Auto.Mode,
                       iManual := "Station_Sys".Manual.Mode,
                       i_ParySensor := 1,
                       iType := 2,
                       i_RunInTimeDelay := T#20S,
                       i_RunOutTimeDelay := T#20S,
                       i_Interlock := "PilzData"."85A2".I6 AND "PilzData"."85A2".I7 AND NOT "PilzData"."85A3".I3,
                       Control := "MotorControl".Dev[17]);
END_REGION

REGION Network 25 (SCL): H-shaftLifting_Motor_OutPut / L-Unloading _LineMotor_OutPut
   "L-Unloading _LineMotor_CW" := "MotorControl".Dev[17].OutControl.o_Start;
   "L-Unloading _LineMotor_CCW" := "MotorControl".Dev[17].OutControl.o_CCWStart OR ("Station_Sys".Auto.Mode AND "AutoProcessControl".Global.L.EmptyPallet);
END_REGION

REGION Network 26: Auto MotorStop
   RUNG wire#powerrail
      Contact( "AlwaysTRUE" )
      wire#w1
      Contact( "Station_Sys".Auto.Mode )
      wire#w2
      Contact( "PilzData"."85A2".I6 )
      Contact( "PilzData"."85A2".I7 )
      Contact( "MotorControl".Dev[17].Auto.Start )
      { S7_Templates := "time_type := Time" } "MotorData".Ton[6].TON(pt := "MotorData"."Time"[6], et =>)
      R_Coil( "MotorControl".Dev[17].Auto.Start )
      R_Coil( "MotorControl".Dev[17].Auto.CCWStart )
   END_RUNG
   RUNG wire#w2
      Contact( "AutoProcessControl".Global.L.EmptyPallet )
      R_Coil( "MotorControl".Dev[17].Auto.Start )
   END_RUNG
   RUNG wire#w1
      { S7_Templates := "SrcType := Time" } LT_Contact(in1 := "MotorData"."Time"[6], in2 := T#1M)
      Move(in := T#1M, out1 => "MotorData"."Time"[6])
   END_RUNG
   // the same network as SCL:
   #_w1 := "AlwaysTRUE" AND "Station_Sys".Auto.Mode;
   "MotorData".Ton[6].TON(IN := #_w1 AND "PilzData"."85A2".I6 AND "PilzData"."85A2".I7 AND "MotorControl".Dev[17].Auto.Start,
                          PT := "MotorData"."Time"[6]);
   IF "MotorData".Ton[6].Q THEN
       "MotorControl".Dev[17].Auto.Start := FALSE;
       "MotorControl".Dev[17].Auto.CCWStart := FALSE;
   END_IF;
   IF #_w1 AND "AutoProcessControl".Global.L.EmptyPallet THEN
       "MotorControl".Dev[17].Auto.Start := FALSE;
   END_IF;
   IF "AlwaysTRUE" AND ("MotorData"."Time"[6] < T#1M) THEN "MotorData"."Time"[6] := T#1M; END_IF;
END_REGION
END_FUNCTION

FUNCTION_BLOCK "MotorContro"   // FB3100, LAD
{ S7_Optimized_Access := 'TRUE' }
// stored: AutoNumber false, MemoryReserve 100, SetENOAutomatically false
   VAR_INPUT
      iAlwaysTrue : Bool;
      iSysRun : Bool;
      iReset : Bool;
      iAuto : Bool;
      iManual : Bool;
      i_ParySensor : Bool;
      i_Alarm : Bool;
      iType : Int;
      i_RunInTimeDelay : Time;
      i_RunOutTimeDelay : Time;
      i_Interlock : Bool;
   END_VAR
   VAR_IN_OUT
      Control : "Motor_Control";
   END_VAR
   VAR
      TON : Array[0..5] of TON_TIME;
      Zero { S7_SetPoint := 'True'} : Array[0..15] of Bool;
   END_VAR
   VAR_TEMP   // added for the SCL form of the ladder/FBD networks
      _w1 : Bool;
   END_VAR
BEGIN

REGION Network 1: Reset
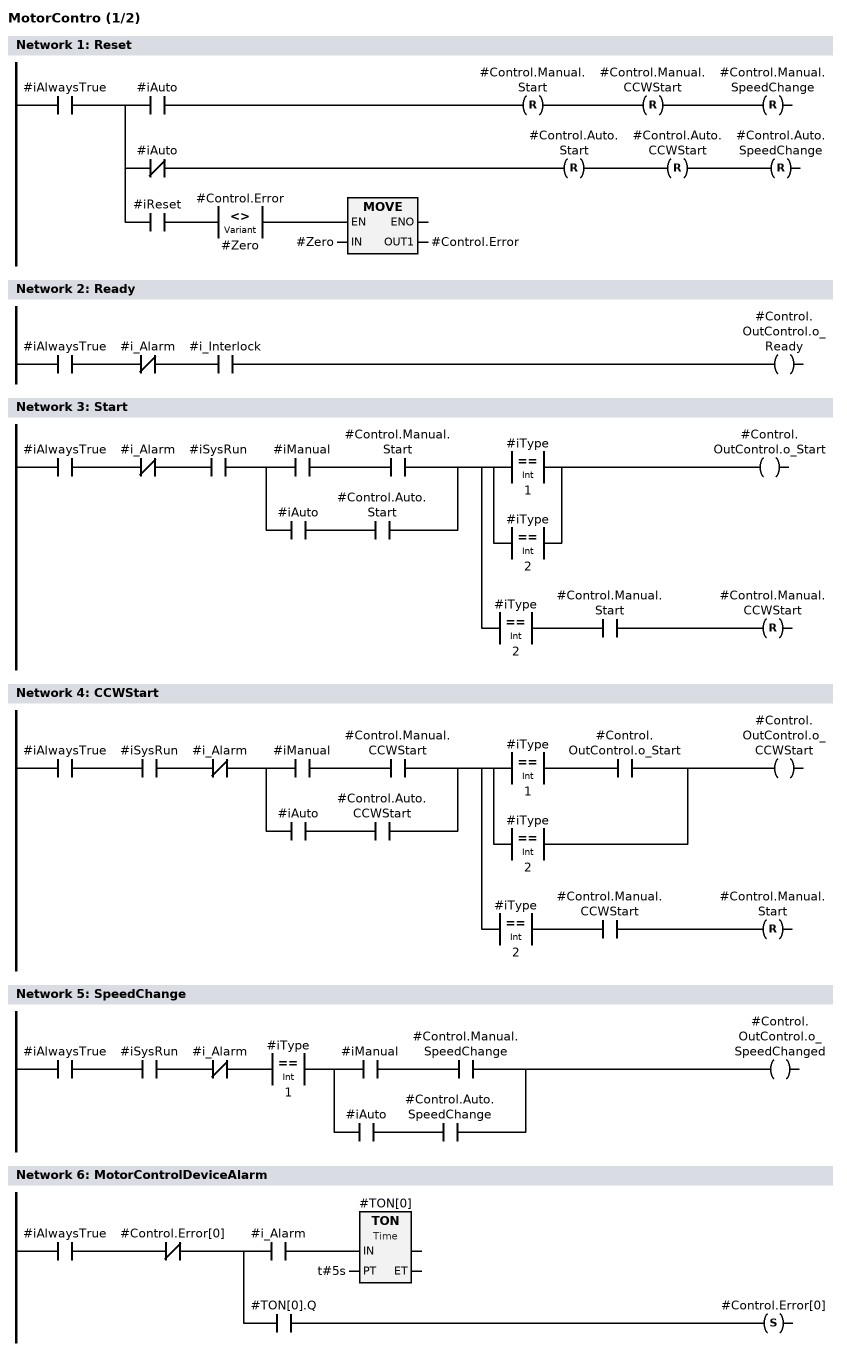
   RUNG wire#powerrail
      Contact( #iAlwaysTrue )
      wire#w1
      Contact( #iAuto )
      R_Coil( #Control.Manual.Start )
      R_Coil( #Control.Manual.CCWStart )
      R_Coil( #Control.Manual.SpeedChange )
   END_RUNG
   RUNG wire#w1
      I_Contact( #iAuto )
      R_Coil( #Control.Auto.Start )
      R_Coil( #Control.Auto.CCWStart )
      R_Coil( #Control.Auto.SpeedChange )
   END_RUNG
   RUNG wire#w1
      Contact( #iReset )
      { S7_Templates := "SrcType := Variant" } NE_Contact(in1 := #Control.Error, in2 := #Zero)
      Move(in := #Zero, out1 => #Control.Error)
   END_RUNG
   // the same network as SCL:
   IF #iAlwaysTrue AND #iAuto THEN
       #Control.Manual.Start := FALSE;
       #Control.Manual.CCWStart := FALSE;
       #Control.Manual.SpeedChange := FALSE;
   END_IF;
   IF #iAlwaysTrue AND NOT #iAuto THEN
       #Control.Auto.Start := FALSE;
       #Control.Auto.CCWStart := FALSE;
       #Control.Auto.SpeedChange := FALSE;
   END_IF;
   IF #iAlwaysTrue AND #iReset AND (#Control.Error <> #Zero) THEN #Control.Error := #Zero; END_IF;
END_REGION

REGION Network 2: Ready
   RUNG wire#powerrail
      Contact( #iAlwaysTrue )
      I_Contact( #i_Alarm )
      Contact( #i_Interlock )
      Coil( #Control.OutControl.o_Ready )
   END_RUNG
   // the same network as SCL:
   #Control.OutControl.o_Ready := #iAlwaysTrue AND NOT #i_Alarm AND #i_Interlock;
END_REGION

REGION Network 3: Start
   RUNG wire#powerrail
      Contact( #iAlwaysTrue )
      I_Contact( #i_Alarm )
      Contact( #iSysRun )
      wire#w1
      Contact( #iManual )
      Contact( #Control.Manual.Start )
      wire#w2
      { S7_Templates := "SrcType := Int" } EQ_Contact(in1 := #iType, in2 := 1)
      wire#w3
      Coil( #Control.OutControl.o_Start )
   END_RUNG
   RUNG wire#w1
      Contact( #iAuto )
      Contact( #Control.Auto.Start )
   END_RUNG wire#w2
   RUNG wire#w2
      { S7_Templates := "SrcType := Int" } EQ_Contact(in1 := #iType, in2 := 2)
   END_RUNG wire#w3
   RUNG wire#w2
      { S7_Templates := "SrcType := Int" } EQ_Contact(in1 := #iType, in2 := 2)
      Contact( #Control.Manual.Start )
      R_Coil( #Control.Manual.CCWStart )
   END_RUNG
   // the same network as SCL:
   #_w1 := #iAlwaysTrue AND NOT #i_Alarm AND #iSysRun AND ((#iManual AND #Control.Manual.Start) OR (#iAuto AND #Control.Auto.Start));
   #Control.OutControl.o_Start := #_w1 AND ((#iType = 1) OR (#iType = 2));
   IF #_w1 AND (#iType = 2) AND #Control.Manual.Start THEN #Control.Manual.CCWStart := FALSE; END_IF;
END_REGION

REGION Network 4: CCWStart
   RUNG wire#powerrail
      Contact( #iAlwaysTrue )
      Contact( #iSysRun )
      I_Contact( #i_Alarm )
      wire#w1
      Contact( #iManual )
      Contact( #Control.Manual.CCWStart )
      wire#w2
      { S7_Templates := "SrcType := Int" } EQ_Contact(in1 := #iType, in2 := 1)
      Contact( #Control.OutControl.o_Start )
      wire#w3
      Coil( #Control.OutControl.o_CCWStart )
   END_RUNG
   RUNG wire#w1
      Contact( #iAuto )
      Contact( #Control.Auto.CCWStart )
   END_RUNG wire#w2
   RUNG wire#w2
      { S7_Templates := "SrcType := Int" } EQ_Contact(in1 := #iType, in2 := 2)
   END_RUNG wire#w3
   RUNG wire#w2
      { S7_Templates := "SrcType := Int" } EQ_Contact(in1 := #iType, in2 := 2)
      Contact( #Control.Manual.CCWStart )
      R_Coil( #Control.Manual.Start )
   END_RUNG
   // the same network as SCL:
   #_w1 := #iAlwaysTrue AND #iSysRun AND NOT #i_Alarm AND ((#iManual AND #Control.Manual.CCWStart) OR (#iAuto AND #Control.Auto.CCWStart));
   #Control.OutControl.o_CCWStart := #_w1 AND (((#iType = 1) AND #Control.OutControl.o_Start) OR (#iType = 2));
   IF #_w1 AND (#iType = 2) AND #Control.Manual.CCWStart THEN #Control.Manual.Start := FALSE; END_IF;
END_REGION

REGION Network 5: SpeedChange
   RUNG wire#powerrail
      Contact( #iAlwaysTrue )
      Contact( #iSysRun )
      I_Contact( #i_Alarm )
      { S7_Templates := "SrcType := Int" } EQ_Contact(in1 := #iType, in2 := 1)
      wire#w1
      Contact( #iManual )
      Contact( #Control.Manual.SpeedChange )
      wire#w2
      Coil( #Control.OutControl.o_SpeedChanged )
   END_RUNG
   RUNG wire#w1
      Contact( #iAuto )
      Contact( #Control.Auto.SpeedChange )
   END_RUNG wire#w2
   // the same network as SCL:
   #Control.OutControl.o_SpeedChanged := #iAlwaysTrue AND #iSysRun AND NOT #i_Alarm AND (#iType = 1) AND ((#iManual AND #Control.Manual.SpeedChange) OR (#iAuto AND #Control.Auto.SpeedChange));
END_REGION

REGION Network 6: MotorControlDeviceAlarm
   RUNG wire#powerrail
      Contact( #iAlwaysTrue )
      I_Contact( #Control.Error[0] )
      wire#w1
      Contact( #i_Alarm )
      { S7_Templates := "time_type := Time" } #TON[0].TON(pt := t#5s, et =>)
   END_RUNG
   RUNG wire#w1
      Contact( #TON[0].Q )
      S_Coil( #Control.Error[0] )
   END_RUNG
   // the same network as SCL:
   #_w1 := #iAlwaysTrue AND NOT #Control.Error[0];
   #TON[0].TON(IN := #_w1 AND #i_Alarm, PT := t#5s);
   IF #_w1 AND #TON[0].Q THEN #Control.Error[0] := TRUE; END_IF;
END_REGION

REGION Network 7: PalletRunInTimeOut
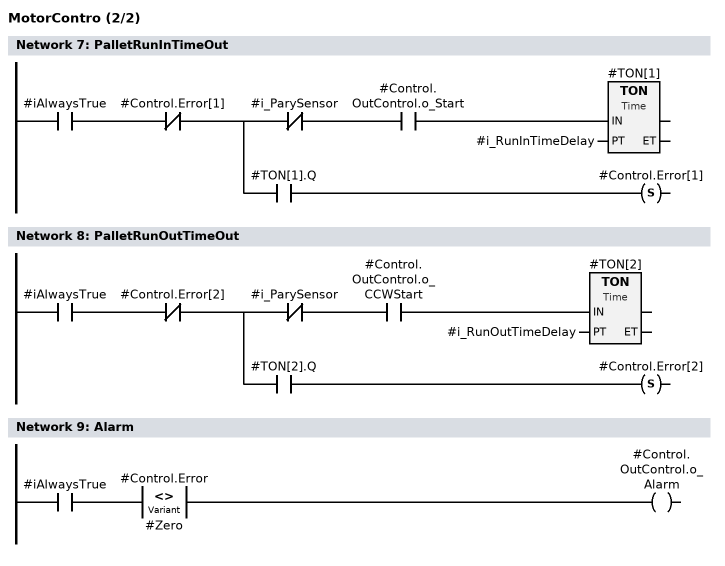
   RUNG wire#powerrail
      Contact( #iAlwaysTrue )
      I_Contact( #Control.Error[1] )
      wire#w1
      I_Contact( #i_ParySensor )
      Contact( #Control.OutControl.o_Start )
      { S7_Templates := "time_type := Time" } #TON[1].TON(pt := #i_RunInTimeDelay, et =>)
   END_RUNG
   RUNG wire#w1
      Contact( #TON[1].Q )
      S_Coil( #Control.Error[1] )
   END_RUNG
   // the same network as SCL:
   #_w1 := #iAlwaysTrue AND NOT #Control.Error[1];
   #TON[1].TON(IN := #_w1 AND NOT #i_ParySensor AND #Control.OutControl.o_Start, PT := #i_RunInTimeDelay);
   IF #_w1 AND #TON[1].Q THEN #Control.Error[1] := TRUE; END_IF;
END_REGION

REGION Network 8: PalletRunOutTimeOut
   RUNG wire#powerrail
      Contact( #iAlwaysTrue )
      I_Contact( #Control.Error[2] )
      wire#w1
      I_Contact( #i_ParySensor )
      Contact( #Control.OutControl.o_CCWStart )
      { S7_Templates := "time_type := Time" } #TON[2].TON(pt := #i_RunOutTimeDelay, et =>)
   END_RUNG
   RUNG wire#w1
      Contact( #TON[2].Q )
      S_Coil( #Control.Error[2] )
   END_RUNG
   // the same network as SCL:
   #_w1 := #iAlwaysTrue AND NOT #Control.Error[2];
   #TON[2].TON(IN := #_w1 AND NOT #i_ParySensor AND #Control.OutControl.o_CCWStart, PT := #i_RunOutTimeDelay);
   IF #_w1 AND #TON[2].Q THEN #Control.Error[2] := TRUE; END_IF;
END_REGION

REGION Network 9: Alarm
   RUNG wire#powerrail
      Contact( #iAlwaysTrue )
      { S7_Templates := "SrcType := Variant" } NE_Contact(in1 := #Control.Error, in2 := #Zero)
      Coil( #Control.OutControl.o_Alarm )
   END_RUNG
   // the same network as SCL:
   #Control.OutControl.o_Alarm := #iAlwaysTrue AND (#Control.Error <> #Zero);
END_REGION
END_FUNCTION_BLOCK

FUNCTION "Stopper" : Void   // FC2600, LAD
{ S7_Optimized_Access := 'TRUE' }
// stored: AutoNumber false, SetENOAutomatically false
BEGIN
END_FUNCTION

FUNCTION "Pilz" : Void   // FC2700, LAD
{ S7_Optimized_Access := 'TRUE' }
// stored: AutoNumber false, SetENOAutomatically false
   VAR_TEMP
      Ret_Val_1 : Int;
      Ret_Val_2 : Int;
      Ret_Val_3 : Int;
      Ret_Val_4 : Int;
   END_VAR
   VAR_TEMP   // added for the SCL form of the ladder/FBD networks
      _w1 : Bool;
   END_VAR
BEGIN

REGION Network 1: 功能块调用 / Pilz
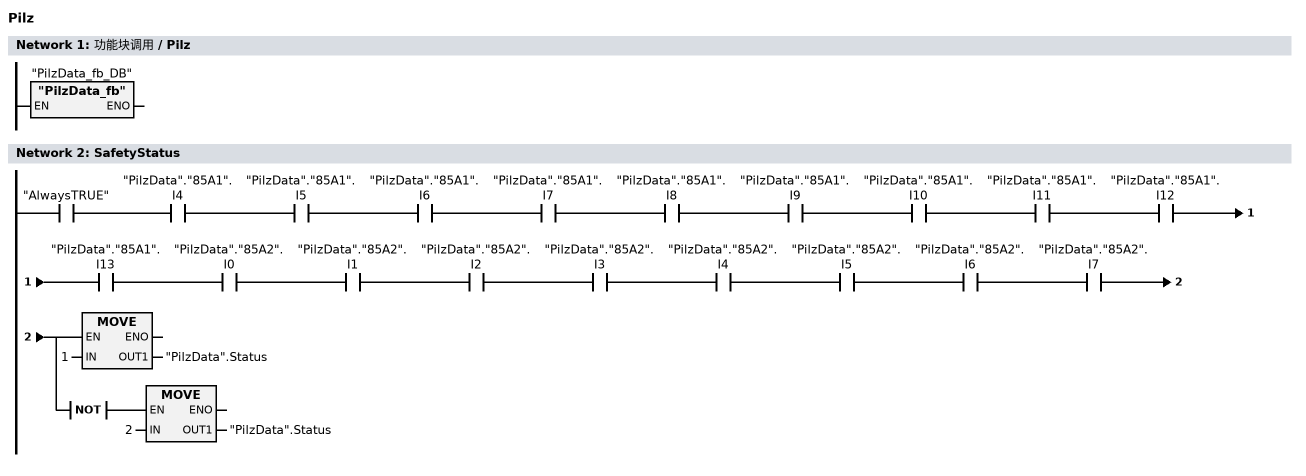
   RUNG wire#powerrail
      "PilzData_fb_DB"()
   END_RUNG
   // the same network as SCL:
   "PilzData_fb_DB"();   // "PilzData_fb"
END_REGION

REGION Network 2: SafetyStatus
   RUNG wire#powerrail
      Contact( "AlwaysTRUE" )
      Contact( "PilzData"."85A1".I4 )
      Contact( "PilzData"."85A1".I5 )
      Contact( "PilzData"."85A1".I6 )
      Contact( "PilzData"."85A1".I7 )
      Contact( "PilzData"."85A1".I8 )
      Contact( "PilzData"."85A1".I9 )
      Contact( "PilzData"."85A1".I10 )
      Contact( "PilzData"."85A1".I11 )
      Contact( "PilzData"."85A1".I12 )
      Contact( "PilzData"."85A1".I13 )
      Contact( "PilzData"."85A2".I0 )
      Contact( "PilzData"."85A2".I1 )
      Contact( "PilzData"."85A2".I2 )
      Contact( "PilzData"."85A2".I3 )
      Contact( "PilzData"."85A2".I4 )
      Contact( "PilzData"."85A2".I5 )
      Contact( "PilzData"."85A2".I6 )
      Contact( "PilzData"."85A2".I7 )
      wire#w1
      Move(in := 1, out1 => "PilzData".Status)
   END_RUNG
   RUNG wire#w1
      Not()
      Move(in := 2, out1 => "PilzData".Status)
   END_RUNG
   // the same network as SCL:
   #_w1 := "AlwaysTRUE" AND "PilzData"."85A1".I4 AND "PilzData"."85A1".I5 AND "PilzData"."85A1".I6 AND "PilzData"."85A1".I7 AND "PilzData"."85A1".I8 AND "PilzData"."85A1".I9 AND "PilzData"."85A1".I10 AND "PilzData"."85A1".I11 AND "PilzData"."85A1".I12 AND "PilzData"."85A1".I13 AND "PilzData"."85A2".I0 AND "PilzData"."85A2".I1 AND "PilzData"."85A2".I2 AND "PilzData"."85A2".I3 AND "PilzData"."85A2".I4 AND "PilzData"."85A2".I5 AND "PilzData"."85A2".I6 AND "PilzData"."85A2".I7;
   IF #_w1 THEN "PilzData".Status := 1; END_IF;
   IF NOT #_w1 THEN "PilzData".Status := 2; END_IF;
END_REGION
END_FUNCTION

FUNCTION "Gluing" : Void   // FC2800, LAD
{ S7_Optimized_Access := 'TRUE' }
// stored: AutoNumber false, SetENOAutomatically false
   VAR_TEMP   // added for the SCL form of the ladder/FBD networks
      _w1 : Bool;
      _w2 : Bool;
   END_VAR
BEGIN

REGION Network 1 (SCL): Input and Output
   //   Input
   "GluingControl".Input.GluingDeviceReady := "iC- GluingDeviceReady";
   "GluingControl".Input.GluingFault := "iC- GluingFault";
   "GluingControl".Input.GluingRefillTank := "iC- GluingRefillTank";
   "GluingControl".Input.GluingTankEmpty := "iC- GluingTankEmpty";

   //   Output
   "oC-GluingPro_X" := "GluingControl".Output.GluingPro_X;
   "oC-GluingPro_Y" := "GluingControl".Output.GluingPro_Y;
   "oC-GluingPro_Z" := "GluingControl".Output.GluingPro_Z;
   "oC-GluingReset" := "GluingControl".Output.GluingReset;
END_REGION

REGION Network 2: Reset
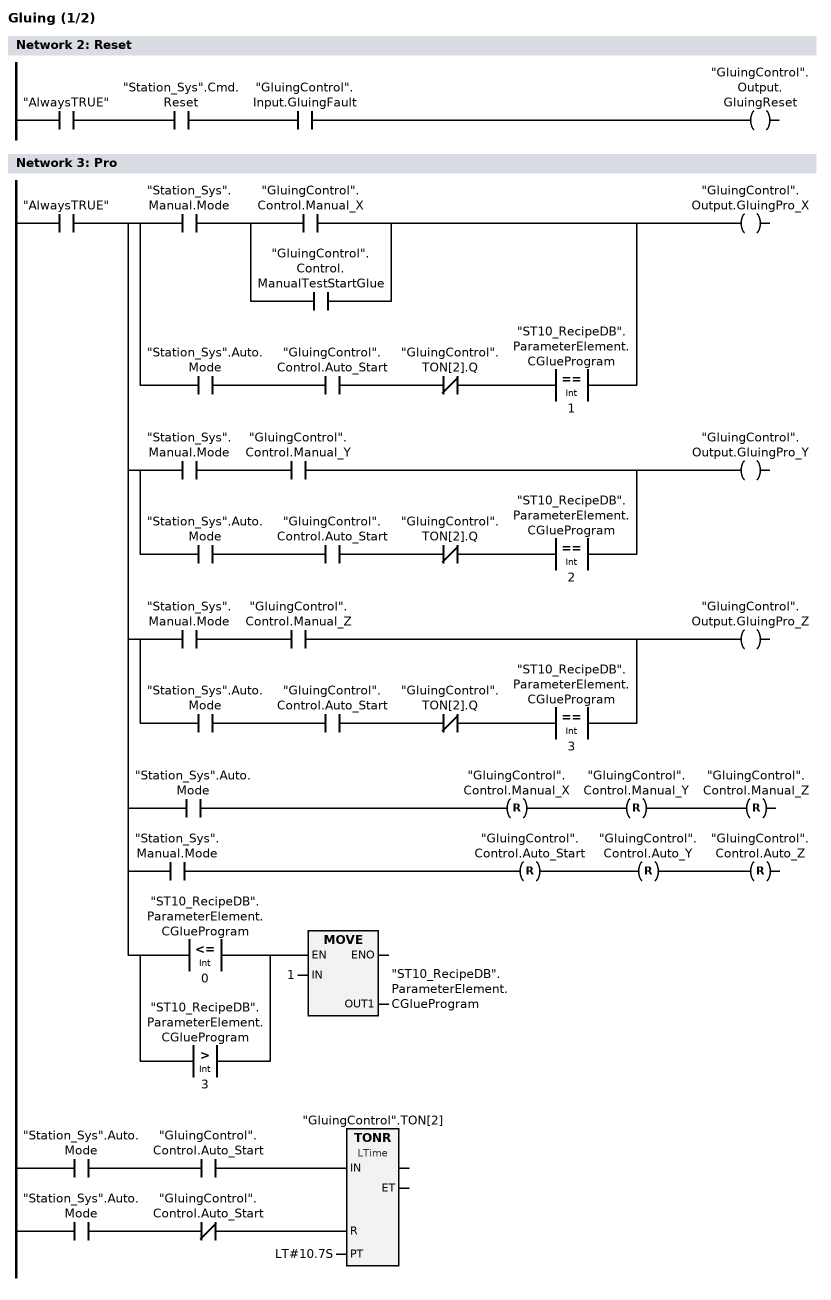
   RUNG wire#powerrail
      Contact( "AlwaysTRUE" )
      Contact( "Station_Sys".Cmd.Reset )
      Contact( "GluingControl".Input.GluingFault )
      Coil( "GluingControl".Output.GluingReset )
   END_RUNG
   // the same network as SCL:
   "GluingControl".Output.GluingReset := "AlwaysTRUE" AND "Station_Sys".Cmd.Reset AND "GluingControl".Input.GluingFault;
END_REGION

REGION Network 3: Pro
   RUNG wire#powerrail
      Contact( "AlwaysTRUE" )
      wire#w1
      Contact( "Station_Sys".Manual.Mode )
      wire#w2
      Contact( "GluingControl".Control.Manual_X )
      wire#w3
      Coil( "GluingControl".Output.GluingPro_X )
   END_RUNG
   RUNG wire#w2
      Contact( "GluingControl".Control.ManualTestStartGlue )
   END_RUNG wire#w3
   RUNG wire#w1
      Contact( "Station_Sys".Auto.Mode )
      Contact( "GluingControl".Control.Auto_Start )
      I_Contact( "GluingControl".TON[2].Q )
      { S7_Templates := "SrcType := Int" } EQ_Contact(in1 := "ST10_RecipeDB".ParameterElement.CGlueProgram, in2 := 1)
   END_RUNG wire#w3
   RUNG wire#w1
      Contact( "Station_Sys".Manual.Mode )
      Contact( "GluingControl".Control.Manual_Y )
      wire#w4
      Coil( "GluingControl".Output.GluingPro_Y )
   END_RUNG
   RUNG wire#w1
      Contact( "Station_Sys".Auto.Mode )
      Contact( "GluingControl".Control.Auto_Start )
      I_Contact( "GluingControl".TON[2].Q )
      { S7_Templates := "SrcType := Int" } EQ_Contact(in1 := "ST10_RecipeDB".ParameterElement.CGlueProgram, in2 := 2)
   END_RUNG wire#w4
   RUNG wire#w1
      Contact( "Station_Sys".Manual.Mode )
      Contact( "GluingControl".Control.Manual_Z )
      wire#w5
      Coil( "GluingControl".Output.GluingPro_Z )
   END_RUNG
   RUNG wire#w1
      Contact( "Station_Sys".Auto.Mode )
      Contact( "GluingControl".Control.Auto_Start )
      I_Contact( "GluingControl".TON[2].Q )
      { S7_Templates := "SrcType := Int" } EQ_Contact(in1 := "ST10_RecipeDB".ParameterElement.CGlueProgram, in2 := 3)
   END_RUNG wire#w5
   RUNG wire#w1
      Contact( "Station_Sys".Auto.Mode )
      R_Coil( "GluingControl".Control.Manual_X )
      R_Coil( "GluingControl".Control.Manual_Y )
      R_Coil( "GluingControl".Control.Manual_Z )
   END_RUNG
   RUNG wire#w1
      Contact( "Station_Sys".Manual.Mode )
      R_Coil( "GluingControl".Control.Auto_Start )
      R_Coil( "GluingControl".Control.Auto_Y )
      R_Coil( "GluingControl".Control.Auto_Z )
   END_RUNG
   RUNG wire#w1
      { S7_Templates := "SrcType := Int" } LE_Contact(in1 := "ST10_RecipeDB".ParameterElement.CGlueProgram, in2 := 0)
      wire#w6
      Move(in := 1, out1 => "ST10_RecipeDB".ParameterElement.CGlueProgram)
   END_RUNG
   RUNG wire#w1
      { S7_Templates := "SrcType := Int" } GT_Contact(in1 := "ST10_RecipeDB".ParameterElement.CGlueProgram, in2 := 3)
   END_RUNG wire#w6
   RUNG wire#powerrail
      Contact( "Station_Sys".Auto.Mode )
      Contact( "GluingControl".Control.Auto_Start )
      { S7_Templates := "time_type := LTime" } "GluingControl".TON[2].TONR(r := wire#w7, pt := LT#10.7S, et =>)
   END_RUNG
   RUNG wire#powerrail
      Contact( "Station_Sys".Auto.Mode )
      I_Contact( "GluingControl".Control.Auto_Start )
   END_RUNG wire#w7
   // the same network as SCL:
   "GluingControl".Output.GluingPro_X := "AlwaysTRUE" AND (("Station_Sys".Manual.Mode AND ("GluingControl".Control.Manual_X OR "GluingControl".Control.ManualTestStartGlue)) OR ("Station_Sys".Auto.Mode AND "GluingControl".Control.Auto_Start AND NOT "GluingControl".TON[2].Q AND ("ST10_RecipeDB".ParameterElement.CGlueProgram = 1)));
   "GluingControl".Output.GluingPro_Y := "AlwaysTRUE" AND (("Station_Sys".Manual.Mode AND "GluingControl".Control.Manual_Y) OR ("Station_Sys".Auto.Mode AND "GluingControl".Control.Auto_Start AND NOT "GluingControl".TON[2].Q AND ("ST10_RecipeDB".ParameterElement.CGlueProgram = 2)));
   "GluingControl".Output.GluingPro_Z := "AlwaysTRUE" AND (("Station_Sys".Manual.Mode AND "GluingControl".Control.Manual_Z) OR ("Station_Sys".Auto.Mode AND "GluingControl".Control.Auto_Start AND NOT "GluingControl".TON[2].Q AND ("ST10_RecipeDB".ParameterElement.CGlueProgram = 3)));
   IF "AlwaysTRUE" AND "Station_Sys".Auto.Mode THEN
       "GluingControl".Control.Manual_X := FALSE;
       "GluingControl".Control.Manual_Y := FALSE;
       "GluingControl".Control.Manual_Z := FALSE;
   END_IF;
   IF "AlwaysTRUE" AND "Station_Sys".Manual.Mode THEN
       "GluingControl".Control.Auto_Start := FALSE;
       "GluingControl".Control.Auto_Y := FALSE;
       "GluingControl".Control.Auto_Z := FALSE;
   END_IF;
   IF "AlwaysTRUE" AND (("ST10_RecipeDB".ParameterElement.CGlueProgram <= 0) OR ("ST10_RecipeDB".ParameterElement.CGlueProgram > 3)) THEN
       "ST10_RecipeDB".ParameterElement.CGlueProgram := 1;
   END_IF;
   "GluingControl".TON[2].TONR(IN := "Station_Sys".Auto.Mode AND "GluingControl".Control.Auto_Start,
                           R := "Station_Sys".Auto.Mode AND NOT "GluingControl".Control.Auto_Start,
                           PT := LT#10.7S);
END_REGION

REGION Network 4: Test
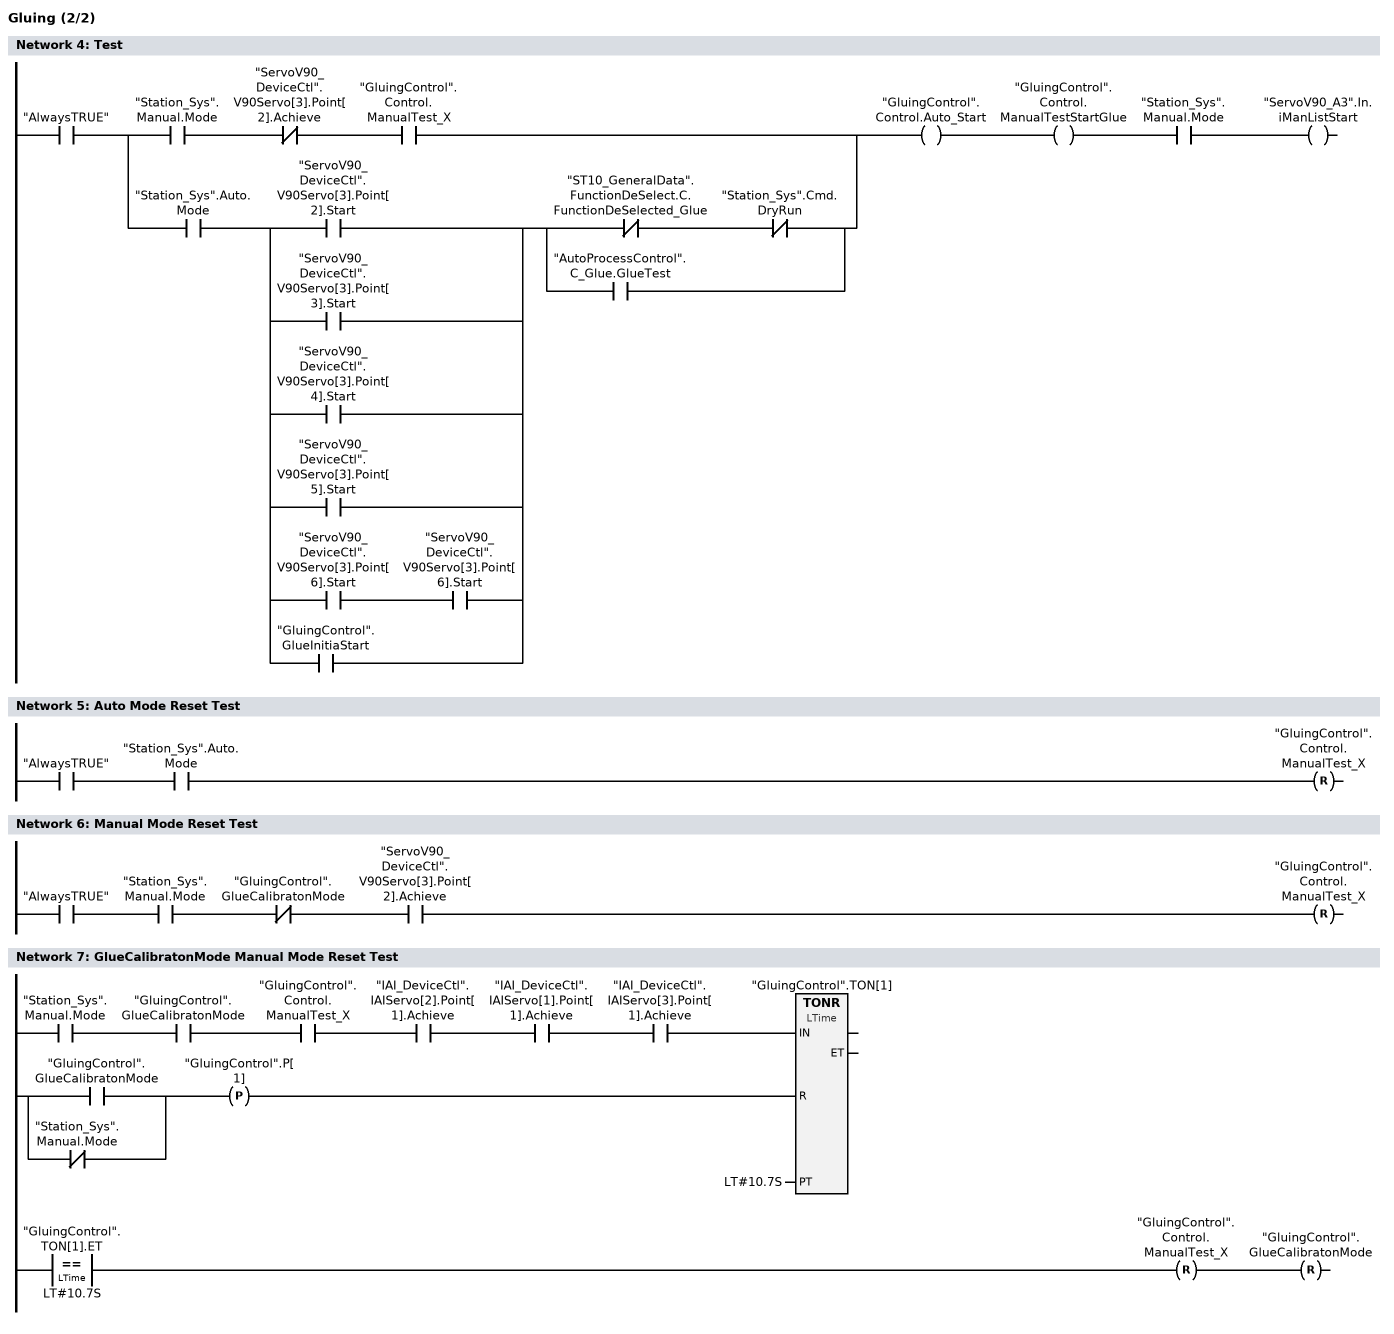
   RUNG wire#powerrail
      Contact( "AlwaysTRUE" )
      wire#w1
      Contact( "Station_Sys".Manual.Mode )
      I_Contact( "ServoV90_DeviceCtl".V90Servo[3].Point[2].Achieve )
      Contact( "GluingControl".Control.ManualTest_X )
      wire#w2
      Coil( "GluingControl".Control.Auto_Start )
      Coil( "GluingControl".Control.ManualTestStartGlue )
      Contact( "Station_Sys".Manual.Mode )
      Coil( "ServoV90_A3".In.iManListStart )
   END_RUNG
   RUNG wire#w1
      Contact( "Station_Sys".Auto.Mode )
      wire#w3
      Contact( "ServoV90_DeviceCtl".V90Servo[3].Point[2].Start )
      wire#w4
      I_Contact( "ST10_GeneralData".FunctionDeSelect.C.FunctionDeSelected_Glue )
      I_Contact( "Station_Sys".Cmd.DryRun )
   END_RUNG wire#w2
   RUNG wire#w3
      Contact( "ServoV90_DeviceCtl".V90Servo[3].Point[3].Start )
   END_RUNG wire#w4
   RUNG wire#w3
      Contact( "ServoV90_DeviceCtl".V90Servo[3].Point[4].Start )
   END_RUNG wire#w4
   RUNG wire#w3
      Contact( "ServoV90_DeviceCtl".V90Servo[3].Point[5].Start )
   END_RUNG wire#w4
   RUNG wire#w3
      Contact( "ServoV90_DeviceCtl".V90Servo[3].Point[6].Start )
      Contact( "ServoV90_DeviceCtl".V90Servo[3].Point[6].Start )
   END_RUNG wire#w4
   RUNG wire#w3
      Contact( "GluingControl".GlueInitiaStart )
   END_RUNG wire#w4
   RUNG wire#w4
      Contact( "AutoProcessControl".C_Glue.GlueTest )
   END_RUNG wire#w2
   // the same network as SCL:
   "GluingControl".Control.Auto_Start := "AlwaysTRUE" AND (("Station_Sys".Manual.Mode AND NOT "ServoV90_DeviceCtl".V90Servo[3].Point[2].Achieve AND "GluingControl".Control.ManualTest_X) OR ("Station_Sys".Auto.Mode AND ("ServoV90_DeviceCtl".V90Servo[3].Point[2].Start OR "ServoV90_DeviceCtl".V90Servo[3].Point[3].Start OR "ServoV90_DeviceCtl".V90Servo[3].Point[4].Start OR "ServoV90_DeviceCtl".V90Servo[3].Point[5].Start OR ("ServoV90_DeviceCtl".V90Servo[3].Point[6].Start AND "ServoV90_DeviceCtl".V90Servo[3].Point[6].Start) OR "GluingControl".GlueInitiaStart) AND ((NOT "ST10_GeneralData".FunctionDeSelect.C.FunctionDeSelected_Glue AND NOT "Station_Sys".Cmd.DryRun) OR "AutoProcessControl".C_Glue.GlueTest)));
   "GluingControl".Control.ManualTestStartGlue := "GluingControl".Control.Auto_Start;
   "ServoV90_A3".In.iManListStart := "GluingControl".Control.Auto_Start AND "Station_Sys".Manual.Mode;
END_REGION

REGION Network 5: Auto Mode Reset Test
   RUNG wire#powerrail
      Contact( "AlwaysTRUE" )
      Contact( "Station_Sys".Auto.Mode )
      R_Coil( "GluingControl".Control.ManualTest_X )
   END_RUNG
   // the same network as SCL:
   IF "AlwaysTRUE" AND "Station_Sys".Auto.Mode THEN "GluingControl".Control.ManualTest_X := FALSE; END_IF;
END_REGION

REGION Network 6: Manual Mode Reset Test
   RUNG wire#powerrail
      Contact( "AlwaysTRUE" )
      Contact( "Station_Sys".Manual.Mode )
      I_Contact( "GluingControl".GlueCalibratonMode )
      Contact( "ServoV90_DeviceCtl".V90Servo[3].Point[2].Achieve )
      R_Coil( "GluingControl".Control.ManualTest_X )
   END_RUNG
   // the same network as SCL:
   IF "AlwaysTRUE" AND "Station_Sys".Manual.Mode AND NOT "GluingControl".GlueCalibratonMode AND "ServoV90_DeviceCtl".V90Servo[3].Point[2].Achieve THEN
       "GluingControl".Control.ManualTest_X := FALSE;
   END_IF;
END_REGION

REGION Network 7: GlueCalibratonMode Manual Mode Reset Test
   RUNG wire#powerrail
      Contact( "Station_Sys".Manual.Mode )
      Contact( "GluingControl".GlueCalibratonMode )
      Contact( "GluingControl".Control.ManualTest_X )
      Contact( "IAI_DeviceCtl".IAIServo[2].Point[1].Achieve )
      Contact( "IAI_DeviceCtl".IAIServo[1].Point[1].Achieve )
      Contact( "IAI_DeviceCtl".IAIServo[3].Point[1].Achieve )
      { S7_Templates := "time_type := LTime" } "GluingControl".TON[1].TONR(r := wire#w2, pt := LT#10.7S, et =>)
   END_RUNG
   RUNG wire#powerrail
      Contact( "GluingControl".GlueCalibratonMode )
      wire#w1
      P_Trig( "GluingControl".P[1] )
   END_RUNG wire#w2
   RUNG wire#powerrail
      I_Contact( "Station_Sys".Manual.Mode )
   END_RUNG wire#w1
   RUNG wire#powerrail
      { S7_Templates := "SrcType := LTime" } EQ_Contact(in1 := "GluingControl".TON[1].ET, in2 := LT#10.7S)
      R_Coil( "GluingControl".Control.ManualTest_X )
      R_Coil( "GluingControl".GlueCalibratonMode )
   END_RUNG
   // the same network as SCL:
   #_w1 := "GluingControl".GlueCalibratonMode OR NOT "Station_Sys".Manual.Mode;
   #_w2 := #_w1 AND NOT "GluingControl".P[1];   // rising edge
   "GluingControl".P[1] := #_w1;
   "GluingControl".TON[1].TONR(IN := "Station_Sys".Manual.Mode AND "GluingControl".GlueCalibratonMode AND "GluingControl".Control.ManualTest_X AND "IAI_DeviceCtl".IAIServo[2].Point[1].Achieve AND "IAI_DeviceCtl".IAIServo[1].Point[1].Achieve AND "IAI_DeviceCtl".IAIServo[3].Point[1].Achieve,
                           R := #_w2,
                           PT := LT#10.7S);
   IF "GluingControl".TON[1].ET = LT#10.7S THEN
       "GluingControl".Control.ManualTest_X := FALSE;
       "GluingControl".GlueCalibratonMode := FALSE;
   END_IF;
END_REGION
END_FUNCTION

FUNCTION "Pallet_NG" : Void   // FC2900, LAD
{ S7_Optimized_Access := 'TRUE' }
// stored: AutoNumber false, SetENOAutomatically false
BEGIN

REGION Network 1
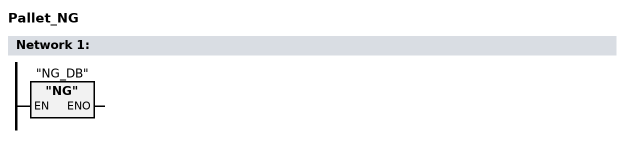
   RUNG wire#powerrail
      "NG_DB"()
   END_RUNG
   // the same network as SCL:
   "NG_DB"();   // "NG"
END_REGION
END_FUNCTION

FUNCTION_BLOCK "NG"   // FB2901, LAD
{ S7_Optimized_Access := 'TRUE' }
// stored: AutoNumber false, MemoryReserve 100, SetENOAutomatically false
   VAR
      NG_L_1 : "NGStatus";
      NG_L_2 { S7_SetPoint := 'True'} : "NGStatus";
      NG_L_3 { S7_SetPoint := 'True'} : "NGStatus";
      NG_UL_1 { S7_SetPoint := 'True'} : "NGStatus";
      NG_UL_2 { S7_SetPoint := 'True'} : "NGStatus";
      NG_UL_3 { S7_SetPoint := 'True'} : "NGStatus";
   END_VAR
   VAR_TEMP   // added for the SCL form of the ladder/FBD networks
      _w1 : Bool;
      _w2 : Bool;
      _w3 : Bool;
      _w4 : Bool;
      _w5 : Bool;
      _w6 : Bool;
      _w7 : Bool;
      _w8 : Bool;
      _w9 : Bool;
      _w10 : Bool;
      _w11 : Bool;
      _w12 : Bool;
      _w13 : Bool;
   END_VAR
BEGIN

REGION Network 1 (SCL): Input
   // NG1
   "PalletNGData".LoadingNGPallet.NG_1_1 := "iE1-UnloadingShaftPressNG_5";
   "PalletNGData".LoadingNGPallet.NG_1_2 := "iE1-UnloadingShaftPressNG_4";
   "PalletNGData".LoadingNGPallet.NG_1_3 := "iE1-UnloadingShaftPressNG_3";
   "PalletNGData".LoadingNGPallet.NG_1_4 := "iE1-UnloadingShaftPressNG_2";
   "PalletNGData".LoadingNGPallet.NG_1_5 := "iE1-UnloadingShaftPressNG_1";

   "PalletNGData".LoadingNGPallet.NG_2_1 := "iE1-UnloadingShaftScanNG_5";
   "PalletNGData".LoadingNGPallet.NG_2_2 := "iE1-UnloadingShaftScanNG_4";
   "PalletNGData".LoadingNGPallet.NG_2_3 := "iE1-UnloadingShaftScanNG_3";
   "PalletNGData".LoadingNGPallet.NG_2_4 := "iE1-UnloadingShaftScanNG_2";
   "PalletNGData".LoadingNGPallet.NG_2_5 := "iE1-UnloadingShaftScanNG_1";

   "PalletNGData".LoadingNGPallet.NG_3_1 := "iE1-UnloadingRingScanNG_5";
   "PalletNGData".LoadingNGPallet.NG_3_2 := "iE1-UnloadingRingScanNG_4";
   "PalletNGData".LoadingNGPallet.NG_3_3 := "iE1-UnloadingRingScanNG_3";
   "PalletNGData".LoadingNGPallet.NG_3_4 := "iE1-UnloadingRingScanNG_2";
   "PalletNGData".LoadingNGPallet.NG_3_5 := "iE1-UnloadingRingScanNG_1";

   // NG2
   "PalletNGData".UnLoadingNGPallet.NG_1_1 := "iE2-UnloadingPressNG_5";
   "PalletNGData".UnLoadingNGPallet.NG_1_2 := "iE2-UnloadingPressNG_4";
   "PalletNGData".UnLoadingNGPallet.NG_1_3 := "iE2-UnloadingPressNG_3";
   "PalletNGData".UnLoadingNGPallet.NG_1_4 := "iE2-UnloadingPressNG_2";
   "PalletNGData".UnLoadingNGPallet.NG_1_5 := "iE2-UnloadingPressNG_1";

   "PalletNGData".UnLoadingNGPallet.NG_2_1 := "iE2-UnloadingMagentScanNG_5";
   "PalletNGData".UnLoadingNGPallet.NG_2_2 := "iE2-UnloadingMagentScanNG_4";
   "PalletNGData".UnLoadingNGPallet.NG_2_3 := "iE2-UnloadingMagentScanNG_3";
   "PalletNGData".UnLoadingNGPallet.NG_2_4 := "iE2-UnloadingMagentScanNG_2";
   "PalletNGData".UnLoadingNGPallet.NG_2_5 := "iE2-UnloadingMagentScanNG_1";

   "PalletNGData".UnLoadingNGPallet.NG_3_1 := "iE2-UnloadingRingScanNG_5";
   "PalletNGData".UnLoadingNGPallet.NG_3_2 := "iE2-UnloadingRingScanNG_4";
   "PalletNGData".UnLoadingNGPallet.NG_3_3 := "iE2-UnloadingRingScanNG_3";
   "PalletNGData".UnLoadingNGPallet.NG_3_4 := "iE2-UnloadingRingScanNG_2";
   "PalletNGData".UnLoadingNGPallet.NG_3_5 := "iE2-UnloadingRingScanNG_1";
END_REGION

REGION Network 2: --------------------------------------- Load -------------------------------------------------------
END_REGION

REGION Network 3: Press
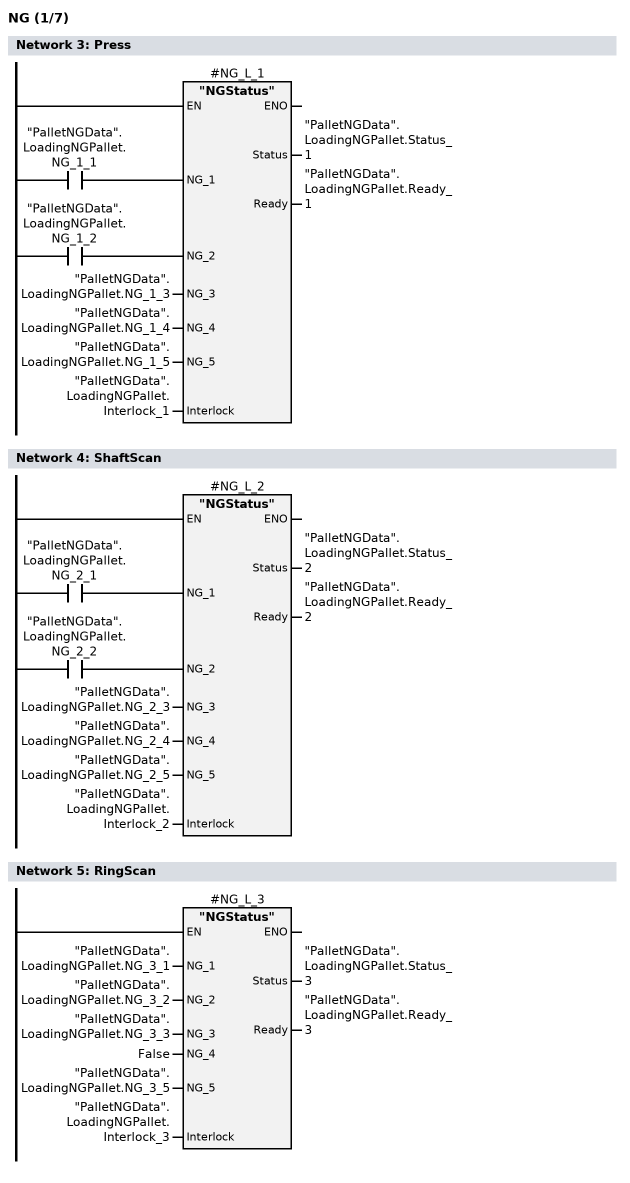
   RUNG wire#powerrail
      #NG_L_1(NG_1 := wire#w1, NG_2 := wire#w2, NG_3 := "PalletNGData".LoadingNGPallet.NG_1_3, NG_4 := "PalletNGData".LoadingNGPallet.NG_1_4, NG_5 := "PalletNGData".LoadingNGPallet.NG_1_5, Interlock := "PalletNGData".LoadingNGPallet.Interlock_1, Status => "PalletNGData".LoadingNGPallet.Status_1, Ready => "PalletNGData".LoadingNGPallet.Ready_1)
   END_RUNG
   RUNG wire#powerrail
      Contact( "PalletNGData".LoadingNGPallet.NG_1_1 )
   END_RUNG wire#w1
   RUNG wire#powerrail
      Contact( "PalletNGData".LoadingNGPallet.NG_1_2 )
   END_RUNG wire#w2
   // the same network as SCL:
   #NG_L_1(NG_1 := "PalletNGData".LoadingNGPallet.NG_1_1,   // "NGStatus"
           NG_2 := "PalletNGData".LoadingNGPallet.NG_1_2,
           NG_3 := "PalletNGData".LoadingNGPallet.NG_1_3,
           NG_4 := "PalletNGData".LoadingNGPallet.NG_1_4,
           NG_5 := "PalletNGData".LoadingNGPallet.NG_1_5,
           Interlock := "PalletNGData".LoadingNGPallet.Interlock_1,
           Status => "PalletNGData".LoadingNGPallet.Status_1,
           Ready => "PalletNGData".LoadingNGPallet.Ready_1);
END_REGION

REGION Network 4: ShaftScan
   RUNG wire#powerrail
      #NG_L_2(NG_1 := wire#w1, NG_2 := wire#w2, NG_3 := "PalletNGData".LoadingNGPallet.NG_2_3, NG_4 := "PalletNGData".LoadingNGPallet.NG_2_4, NG_5 := "PalletNGData".LoadingNGPallet.NG_2_5, Interlock := "PalletNGData".LoadingNGPallet.Interlock_2, Status => "PalletNGData".LoadingNGPallet.Status_2, Ready => "PalletNGData".LoadingNGPallet.Ready_2)
   END_RUNG
   RUNG wire#powerrail
      Contact( "PalletNGData".LoadingNGPallet.NG_2_1 )
   END_RUNG wire#w1
   RUNG wire#powerrail
      Contact( "PalletNGData".LoadingNGPallet.NG_2_2 )
   END_RUNG wire#w2
   // the same network as SCL:
   #NG_L_2(NG_1 := "PalletNGData".LoadingNGPallet.NG_2_1,   // "NGStatus"
           NG_2 := "PalletNGData".LoadingNGPallet.NG_2_2,
           NG_3 := "PalletNGData".LoadingNGPallet.NG_2_3,
           NG_4 := "PalletNGData".LoadingNGPallet.NG_2_4,
           NG_5 := "PalletNGData".LoadingNGPallet.NG_2_5,
           Interlock := "PalletNGData".LoadingNGPallet.Interlock_2,
           Status => "PalletNGData".LoadingNGPallet.Status_2,
           Ready => "PalletNGData".LoadingNGPallet.Ready_2);
END_REGION

REGION Network 5: RingScan
   RUNG wire#powerrail
      #NG_L_3(NG_1 := "PalletNGData".LoadingNGPallet.NG_3_1, NG_2 := "PalletNGData".LoadingNGPallet.NG_3_2, NG_3 := "PalletNGData".LoadingNGPallet.NG_3_3, NG_4 := False, NG_5 := "PalletNGData".LoadingNGPallet.NG_3_5, Interlock := "PalletNGData".LoadingNGPallet.Interlock_3, Status => "PalletNGData".LoadingNGPallet.Status_3, Ready => "PalletNGData".LoadingNGPallet.Ready_3)
   END_RUNG
   // the same network as SCL:
   #NG_L_3(NG_1 := "PalletNGData".LoadingNGPallet.NG_3_1,   // "NGStatus"
           NG_2 := "PalletNGData".LoadingNGPallet.NG_3_2,
           NG_3 := "PalletNGData".LoadingNGPallet.NG_3_3,
           NG_4 := False,
           NG_5 := "PalletNGData".LoadingNGPallet.NG_3_5,
           Interlock := "PalletNGData".LoadingNGPallet.Interlock_3,
           Status => "PalletNGData".LoadingNGPallet.Status_3,
           Ready => "PalletNGData".LoadingNGPallet.Ready_3);
END_REGION

REGION Network 6: InterLock
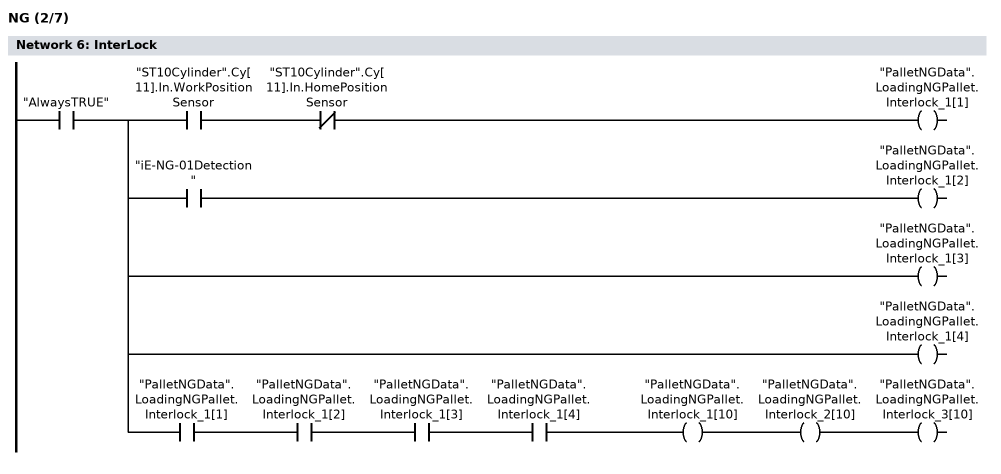
   RUNG wire#powerrail
      Contact( "AlwaysTRUE" )
      wire#w1
      Contact( "ST10Cylinder".Cy[11].In.WorkPositionSensor )
      I_Contact( "ST10Cylinder".Cy[11].In.HomePositionSensor )
      Coil( "PalletNGData".LoadingNGPallet.Interlock_1[1] )
   END_RUNG
   RUNG wire#w1
      Contact( "iE-NG-01Detection" )
      Coil( "PalletNGData".LoadingNGPallet.Interlock_1[2] )
   END_RUNG
   RUNG wire#w1
      Coil( "PalletNGData".LoadingNGPallet.Interlock_1[3] )
   END_RUNG
   RUNG wire#w1
      Coil( "PalletNGData".LoadingNGPallet.Interlock_1[4] )
   END_RUNG
   RUNG wire#w1
      Contact( "PalletNGData".LoadingNGPallet.Interlock_1[1] )
      Contact( "PalletNGData".LoadingNGPallet.Interlock_1[2] )
      Contact( "PalletNGData".LoadingNGPallet.Interlock_1[3] )
      Contact( "PalletNGData".LoadingNGPallet.Interlock_1[4] )
      Coil( "PalletNGData".LoadingNGPallet.Interlock_1[10] )
      Coil( "PalletNGData".LoadingNGPallet.Interlock_2[10] )
      Coil( "PalletNGData".LoadingNGPallet.Interlock_3[10] )
   END_RUNG
   // the same network as SCL:
   "PalletNGData".LoadingNGPallet.Interlock_1[1] := "AlwaysTRUE" AND "ST10Cylinder".Cy[11].In.WorkPositionSensor AND NOT "ST10Cylinder".Cy[11].In.HomePositionSensor;
   "PalletNGData".LoadingNGPallet.Interlock_1[2] := "AlwaysTRUE" AND "iE-NG-01Detection";
   "PalletNGData".LoadingNGPallet.Interlock_1[3] := "AlwaysTRUE";
   "PalletNGData".LoadingNGPallet.Interlock_1[4] := "AlwaysTRUE";
   #_w1 := "AlwaysTRUE" AND "PalletNGData".LoadingNGPallet.Interlock_1[1] AND "PalletNGData".LoadingNGPallet.Interlock_1[2] AND "PalletNGData".LoadingNGPallet.Interlock_1[3] AND "PalletNGData".LoadingNGPallet.Interlock_1[4];
   "PalletNGData".LoadingNGPallet.Interlock_1[10] := #_w1;
   "PalletNGData".LoadingNGPallet.Interlock_2[10] := #_w1;
   "PalletNGData".LoadingNGPallet.Interlock_3[10] := #_w1;
END_REGION

REGION Network 7: NG_Button
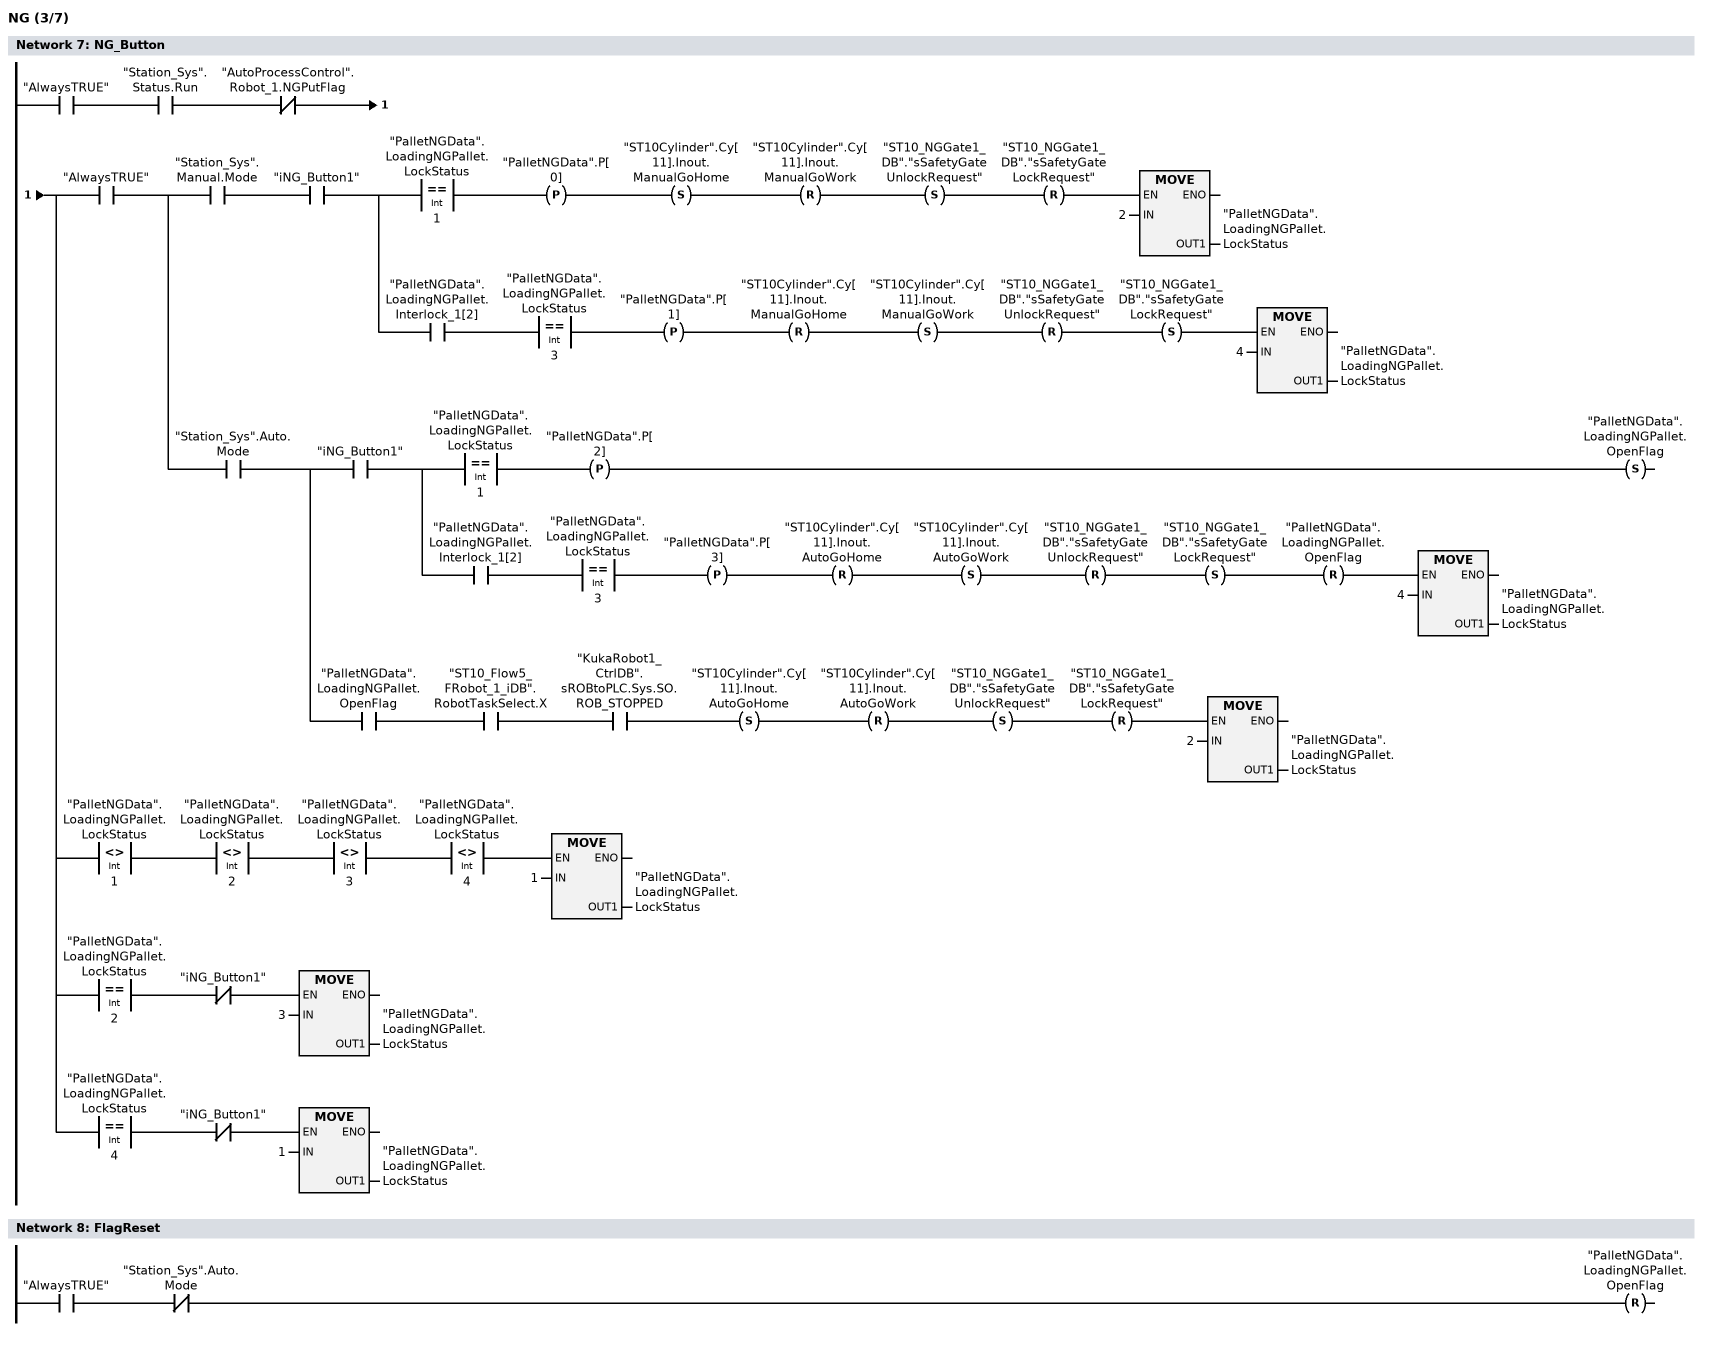
   RUNG wire#powerrail
      Contact( "AlwaysTRUE" )
      Contact( "Station_Sys".Status.Run )
      I_Contact( "AutoProcessControl".Robot_1.NGPutFlag )
      wire#w1
      Contact( "AlwaysTRUE" )
      wire#w2
      Contact( "Station_Sys".Manual.Mode )
      Contact( "iNG_Button1" )
      wire#w3
      { S7_Templates := "SrcType := Int" } EQ_Contact(in1 := "PalletNGData".LoadingNGPallet.LockStatus, in2 := 1)
      P_Trig( "PalletNGData".P[0] )
      S_Coil( "ST10Cylinder".Cy[11].Inout.ManualGoHome )
      R_Coil( "ST10Cylinder".Cy[11].Inout.ManualGoWork )
      S_Coil( "ST10_NGGate1_DB"."sSafetyGate UnlockRequest" )
      R_Coil( "ST10_NGGate1_DB"."sSafetyGate LockRequest" )
      Move(in := 2, out1 => "PalletNGData".LoadingNGPallet.LockStatus)
   END_RUNG
   RUNG wire#w3
      Contact( "PalletNGData".LoadingNGPallet.Interlock_1[2] )
      { S7_Templates := "SrcType := Int" } EQ_Contact(in1 := "PalletNGData".LoadingNGPallet.LockStatus, in2 := 3)
      P_Trig( "PalletNGData".P[1] )
      R_Coil( "ST10Cylinder".Cy[11].Inout.ManualGoHome )
      S_Coil( "ST10Cylinder".Cy[11].Inout.ManualGoWork )
      R_Coil( "ST10_NGGate1_DB"."sSafetyGate UnlockRequest" )
      S_Coil( "ST10_NGGate1_DB"."sSafetyGate LockRequest" )
      Move(in := 4, out1 => "PalletNGData".LoadingNGPallet.LockStatus)
   END_RUNG
   RUNG wire#w2
      Contact( "Station_Sys".Auto.Mode )
      wire#w4
      Contact( "iNG_Button1" )
      wire#w5
      { S7_Templates := "SrcType := Int" } EQ_Contact(in1 := "PalletNGData".LoadingNGPallet.LockStatus, in2 := 1)
      P_Trig( "PalletNGData".P[2] )
      S_Coil( "PalletNGData".LoadingNGPallet.OpenFlag )
   END_RUNG
   RUNG wire#w5
      Contact( "PalletNGData".LoadingNGPallet.Interlock_1[2] )
      { S7_Templates := "SrcType := Int" } EQ_Contact(in1 := "PalletNGData".LoadingNGPallet.LockStatus, in2 := 3)
      P_Trig( "PalletNGData".P[3] )
      R_Coil( "ST10Cylinder".Cy[11].Inout.AutoGoHome )
      S_Coil( "ST10Cylinder".Cy[11].Inout.AutoGoWork )
      R_Coil( "ST10_NGGate1_DB"."sSafetyGate UnlockRequest" )
      S_Coil( "ST10_NGGate1_DB"."sSafetyGate LockRequest" )
      R_Coil( "PalletNGData".LoadingNGPallet.OpenFlag )
      Move(in := 4, out1 => "PalletNGData".LoadingNGPallet.LockStatus)
   END_RUNG
   RUNG wire#w4
      Contact( "PalletNGData".LoadingNGPallet.OpenFlag )
      Contact( "ST10_Flow5_FRobot_1_iDB".RobotTaskSelect.X )
      Contact( "KukaRobot1_CtrlDB".sROBtoPLC.Sys.SO.ROB_STOPPED )
      S_Coil( "ST10Cylinder".Cy[11].Inout.AutoGoHome )
      R_Coil( "ST10Cylinder".Cy[11].Inout.AutoGoWork )
      S_Coil( "ST10_NGGate1_DB"."sSafetyGate UnlockRequest" )
      R_Coil( "ST10_NGGate1_DB"."sSafetyGate LockRequest" )
      Move(in := 2, out1 => "PalletNGData".LoadingNGPallet.LockStatus)
   END_RUNG
   RUNG wire#w1
      { S7_Templates := "SrcType := Int" } NE_Contact(in1 := "PalletNGData".LoadingNGPallet.LockStatus, in2 := 1)
      { S7_Templates := "SrcType := Int" } NE_Contact(in1 := "PalletNGData".LoadingNGPallet.LockStatus, in2 := 2)
      { S7_Templates := "SrcType := Int" } NE_Contact(in1 := "PalletNGData".LoadingNGPallet.LockStatus, in2 := 3)
      { S7_Templates := "SrcType := Int" } NE_Contact(in1 := "PalletNGData".LoadingNGPallet.LockStatus, in2 := 4)
      Move(in := 1, out1 => "PalletNGData".LoadingNGPallet.LockStatus)
   END_RUNG
   RUNG wire#w1
      { S7_Templates := "SrcType := Int" } EQ_Contact(in1 := "PalletNGData".LoadingNGPallet.LockStatus, in2 := 2)
      I_Contact( "iNG_Button1" )
      Move(in := 3, out1 => "PalletNGData".LoadingNGPallet.LockStatus)
   END_RUNG
   RUNG wire#w1
      { S7_Templates := "SrcType := Int" } EQ_Contact(in1 := "PalletNGData".LoadingNGPallet.LockStatus, in2 := 4)
      I_Contact( "iNG_Button1" )
      Move(in := 1, out1 => "PalletNGData".LoadingNGPallet.LockStatus)
   END_RUNG
   // the same network as SCL:
   #_w1 := "AlwaysTRUE" AND "Station_Sys".Status.Run AND NOT "AutoProcessControl".Robot_1.NGPutFlag;
   #_w2 := #_w1 AND "AlwaysTRUE";
   #_w3 := #_w2 AND "Station_Sys".Manual.Mode AND "iNG_Button1";
   #_w4 := #_w3 AND ("PalletNGData".LoadingNGPallet.LockStatus = 1);
   #_w5 := #_w4 AND NOT "PalletNGData".P[0];   // rising edge
   "PalletNGData".P[0] := #_w4;
   IF #_w5 THEN
       "ST10Cylinder".Cy[11].Inout.ManualGoHome := TRUE;
       "ST10Cylinder".Cy[11].Inout.ManualGoWork := FALSE;
       "ST10_NGGate1_DB"."sSafetyGate UnlockRequest" := TRUE;
       "ST10_NGGate1_DB"."sSafetyGate LockRequest" := FALSE;
       "PalletNGData".LoadingNGPallet.LockStatus := 2;
   END_IF;
   #_w6 := #_w3 AND "PalletNGData".LoadingNGPallet.Interlock_1[2] AND ("PalletNGData".LoadingNGPallet.LockStatus = 3);
   #_w7 := #_w6 AND NOT "PalletNGData".P[1];   // rising edge
   "PalletNGData".P[1] := #_w6;
   IF #_w7 THEN
       "ST10Cylinder".Cy[11].Inout.ManualGoHome := FALSE;
       "ST10Cylinder".Cy[11].Inout.ManualGoWork := TRUE;
       "ST10_NGGate1_DB"."sSafetyGate UnlockRequest" := FALSE;
       "ST10_NGGate1_DB"."sSafetyGate LockRequest" := TRUE;
       "PalletNGData".LoadingNGPallet.LockStatus := 4;
   END_IF;
   #_w8 := #_w2 AND "Station_Sys".Auto.Mode;
   #_w9 := #_w8 AND "iNG_Button1";
   #_w10 := #_w9 AND ("PalletNGData".LoadingNGPallet.LockStatus = 1);
   #_w11 := #_w10 AND NOT "PalletNGData".P[2];   // rising edge
   "PalletNGData".P[2] := #_w10;
   IF #_w11 THEN "PalletNGData".LoadingNGPallet.OpenFlag := TRUE; END_IF;
   #_w12 := #_w9 AND "PalletNGData".LoadingNGPallet.Interlock_1[2] AND ("PalletNGData".LoadingNGPallet.LockStatus = 3);
   #_w13 := #_w12 AND NOT "PalletNGData".P[3];   // rising edge
   "PalletNGData".P[3] := #_w12;
   IF #_w13 THEN
       "ST10Cylinder".Cy[11].Inout.AutoGoHome := FALSE;
       "ST10Cylinder".Cy[11].Inout.AutoGoWork := TRUE;
       "ST10_NGGate1_DB"."sSafetyGate UnlockRequest" := FALSE;
       "ST10_NGGate1_DB"."sSafetyGate LockRequest" := TRUE;
       "PalletNGData".LoadingNGPallet.OpenFlag := FALSE;
       "PalletNGData".LoadingNGPallet.LockStatus := 4;
   END_IF;
   IF #_w8 AND "PalletNGData".LoadingNGPallet.OpenFlag AND "ST10_Flow5_FRobot_1_iDB".RobotTaskSelect.X AND "KukaRobot1_CtrlDB".sROBtoPLC.Sys.SO.ROB_STOPPED THEN
       "ST10Cylinder".Cy[11].Inout.AutoGoHome := TRUE;
       "ST10Cylinder".Cy[11].Inout.AutoGoWork := FALSE;
       "ST10_NGGate1_DB"."sSafetyGate UnlockRequest" := TRUE;
       "ST10_NGGate1_DB"."sSafetyGate LockRequest" := FALSE;
       "PalletNGData".LoadingNGPallet.LockStatus := 2;
   END_IF;
   IF #_w1 AND ("PalletNGData".LoadingNGPallet.LockStatus <> 1) AND ("PalletNGData".LoadingNGPallet.LockStatus <> 2) AND ("PalletNGData".LoadingNGPallet.LockStatus <> 3) AND ("PalletNGData".LoadingNGPallet.LockStatus <> 4) THEN
       "PalletNGData".LoadingNGPallet.LockStatus := 1;
   END_IF;
   IF #_w1 AND ("PalletNGData".LoadingNGPallet.LockStatus = 2) AND NOT "iNG_Button1" THEN
       "PalletNGData".LoadingNGPallet.LockStatus := 3;
   END_IF;
   IF #_w1 AND ("PalletNGData".LoadingNGPallet.LockStatus = 4) AND NOT "iNG_Button1" THEN
       "PalletNGData".LoadingNGPallet.LockStatus := 1;
   END_IF;
END_REGION

REGION Network 8: FlagReset
   RUNG wire#powerrail
      Contact( "AlwaysTRUE" )
      I_Contact( "Station_Sys".Auto.Mode )
      R_Coil( "PalletNGData".LoadingNGPallet.OpenFlag )
   END_RUNG
   // the same network as SCL:
   IF "AlwaysTRUE" AND NOT "Station_Sys".Auto.Mode THEN
       "PalletNGData".LoadingNGPallet.OpenFlag := FALSE;
   END_IF;
END_REGION

REGION Network 9: NG Door
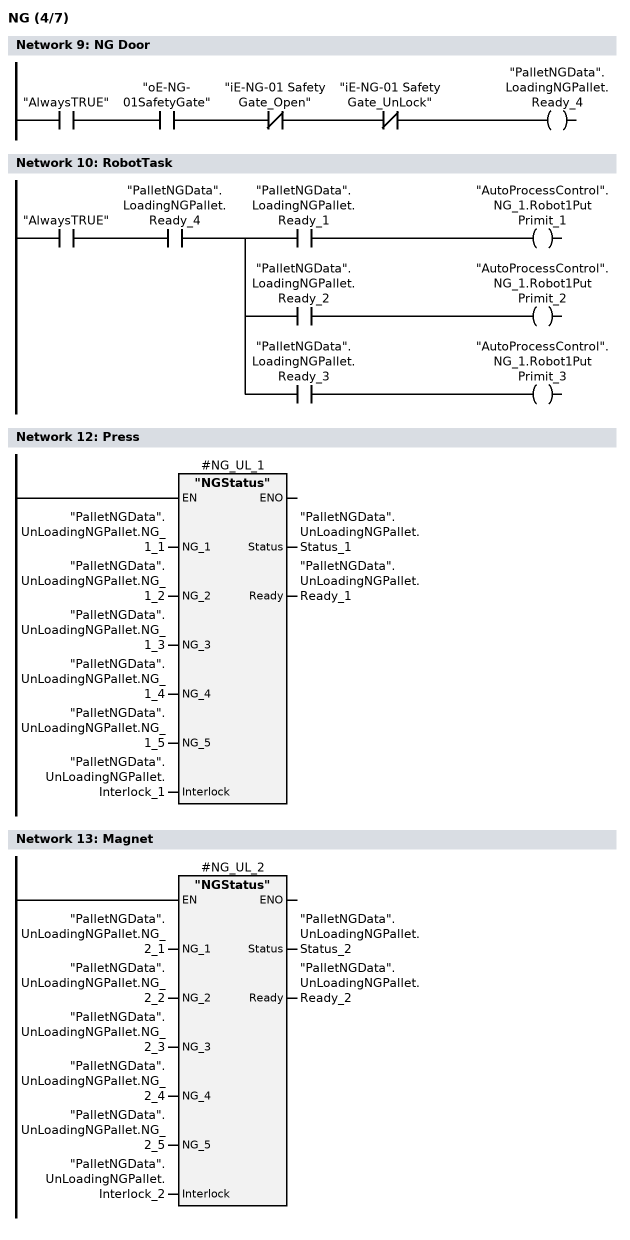
   RUNG wire#powerrail
      Contact( "AlwaysTRUE" )
      Contact( "oE-NG-01SafetyGate" )
      I_Contact( "iE-NG-01 Safety Gate_Open" )
      I_Contact( "iE-NG-01 Safety Gate_UnLock" )
      Coil( "PalletNGData".LoadingNGPallet.Ready_4 )
   END_RUNG
   // the same network as SCL:
   "PalletNGData".LoadingNGPallet.Ready_4 := "AlwaysTRUE" AND "oE-NG-01SafetyGate" AND NOT "iE-NG-01 Safety Gate_Open" AND NOT "iE-NG-01 Safety Gate_UnLock";
END_REGION

REGION Network 10: RobotTask
   RUNG wire#powerrail
      Contact( "AlwaysTRUE" )
      Contact( "PalletNGData".LoadingNGPallet.Ready_4 )
      wire#w1
      Contact( "PalletNGData".LoadingNGPallet.Ready_1 )
      Coil( "AutoProcessControl".NG_1.Robot1PutPrimit_1 )
   END_RUNG
   RUNG wire#w1
      Contact( "PalletNGData".LoadingNGPallet.Ready_2 )
      Coil( "AutoProcessControl".NG_1.Robot1PutPrimit_2 )
   END_RUNG
   RUNG wire#w1
      Contact( "PalletNGData".LoadingNGPallet.Ready_3 )
      Coil( "AutoProcessControl".NG_1.Robot1PutPrimit_3 )
   END_RUNG
   // the same network as SCL:
   #_w1 := "AlwaysTRUE" AND "PalletNGData".LoadingNGPallet.Ready_4;
   "AutoProcessControl".NG_1.Robot1PutPrimit_1 := #_w1 AND "PalletNGData".LoadingNGPallet.Ready_1;
   "AutoProcessControl".NG_1.Robot1PutPrimit_2 := #_w1 AND "PalletNGData".LoadingNGPallet.Ready_2;
   "AutoProcessControl".NG_1.Robot1PutPrimit_3 := #_w1 AND "PalletNGData".LoadingNGPallet.Ready_3;
END_REGION

REGION Network 11: --------------------------------------- UnLoad -------------------------------------------------------
END_REGION

REGION Network 12: Press
   RUNG wire#powerrail
      #NG_UL_1(NG_1 := "PalletNGData".UnLoadingNGPallet.NG_1_1, NG_2 := "PalletNGData".UnLoadingNGPallet.NG_1_2, NG_3 := "PalletNGData".UnLoadingNGPallet.NG_1_3, NG_4 := "PalletNGData".UnLoadingNGPallet.NG_1_4, NG_5 := "PalletNGData".UnLoadingNGPallet.NG_1_5, Interlock := "PalletNGData".UnLoadingNGPallet.Interlock_1, Status => "PalletNGData".UnLoadingNGPallet.Status_1, Ready => "PalletNGData".UnLoadingNGPallet.Ready_1)
   END_RUNG
   // the same network as SCL:
   #NG_UL_1(NG_1 := "PalletNGData".UnLoadingNGPallet.NG_1_1,   // "NGStatus"
            NG_2 := "PalletNGData".UnLoadingNGPallet.NG_1_2,
            NG_3 := "PalletNGData".UnLoadingNGPallet.NG_1_3,
            NG_4 := "PalletNGData".UnLoadingNGPallet.NG_1_4,
            NG_5 := "PalletNGData".UnLoadingNGPallet.NG_1_5,
            Interlock := "PalletNGData".UnLoadingNGPallet.Interlock_1,
            Status => "PalletNGData".UnLoadingNGPallet.Status_1,
            Ready => "PalletNGData".UnLoadingNGPallet.Ready_1);
END_REGION

REGION Network 13: Magnet
   RUNG wire#powerrail
      #NG_UL_2(NG_1 := "PalletNGData".UnLoadingNGPallet.NG_2_1, NG_2 := "PalletNGData".UnLoadingNGPallet.NG_2_2, NG_3 := "PalletNGData".UnLoadingNGPallet.NG_2_3, NG_4 := "PalletNGData".UnLoadingNGPallet.NG_2_4, NG_5 := "PalletNGData".UnLoadingNGPallet.NG_2_5, Interlock := "PalletNGData".UnLoadingNGPallet.Interlock_2, Status => "PalletNGData".UnLoadingNGPallet.Status_2, Ready => "PalletNGData".UnLoadingNGPallet.Ready_2)
   END_RUNG
   // the same network as SCL:
   #NG_UL_2(NG_1 := "PalletNGData".UnLoadingNGPallet.NG_2_1,   // "NGStatus"
            NG_2 := "PalletNGData".UnLoadingNGPallet.NG_2_2,
            NG_3 := "PalletNGData".UnLoadingNGPallet.NG_2_3,
            NG_4 := "PalletNGData".UnLoadingNGPallet.NG_2_4,
            NG_5 := "PalletNGData".UnLoadingNGPallet.NG_2_5,
            Interlock := "PalletNGData".UnLoadingNGPallet.Interlock_2,
            Status => "PalletNGData".UnLoadingNGPallet.Status_2,
            Ready => "PalletNGData".UnLoadingNGPallet.Ready_2);
END_REGION

REGION Network 14: Ring
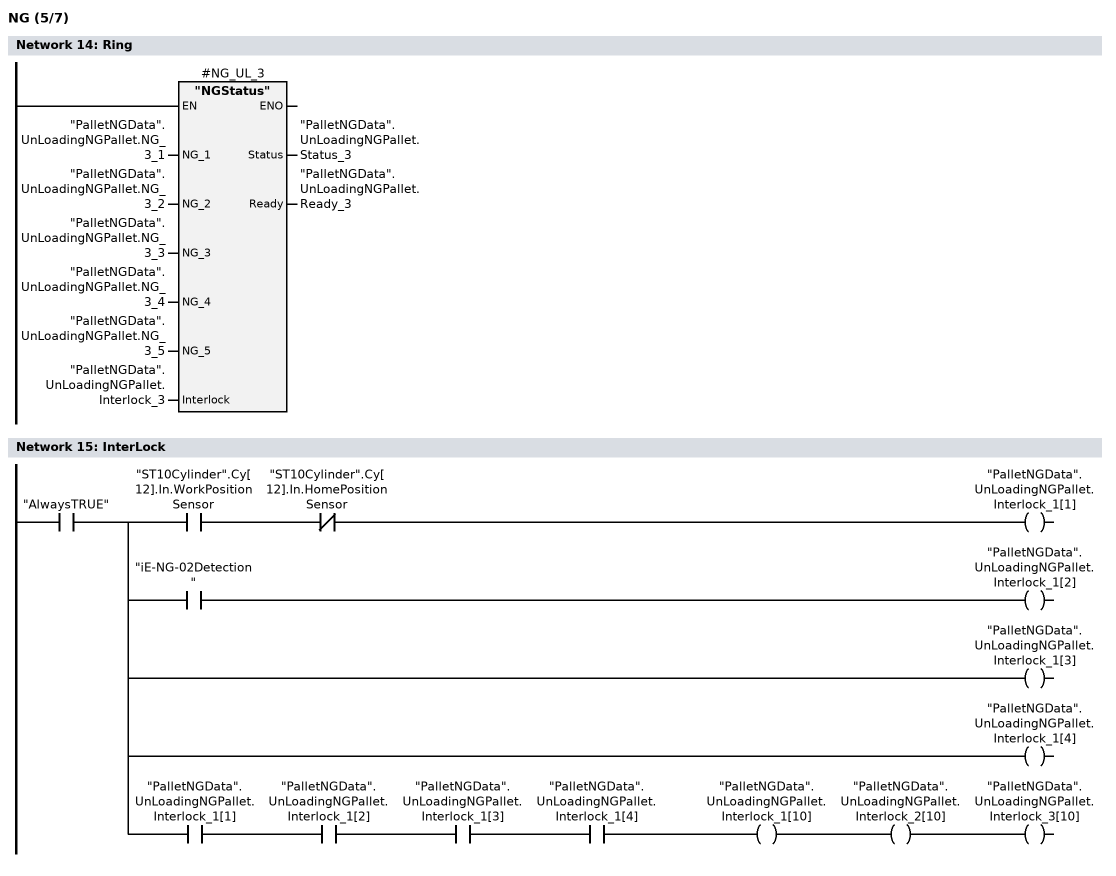
   RUNG wire#powerrail
      #NG_UL_3(NG_1 := "PalletNGData".UnLoadingNGPallet.NG_3_1, NG_2 := "PalletNGData".UnLoadingNGPallet.NG_3_2, NG_3 := "PalletNGData".UnLoadingNGPallet.NG_3_3, NG_4 := "PalletNGData".UnLoadingNGPallet.NG_3_4, NG_5 := "PalletNGData".UnLoadingNGPallet.NG_3_5, Interlock := "PalletNGData".UnLoadingNGPallet.Interlock_3, Status => "PalletNGData".UnLoadingNGPallet.Status_3, Ready => "PalletNGData".UnLoadingNGPallet.Ready_3)
   END_RUNG
   // the same network as SCL:
   #NG_UL_3(NG_1 := "PalletNGData".UnLoadingNGPallet.NG_3_1,   // "NGStatus"
            NG_2 := "PalletNGData".UnLoadingNGPallet.NG_3_2,
            NG_3 := "PalletNGData".UnLoadingNGPallet.NG_3_3,
            NG_4 := "PalletNGData".UnLoadingNGPallet.NG_3_4,
            NG_5 := "PalletNGData".UnLoadingNGPallet.NG_3_5,
            Interlock := "PalletNGData".UnLoadingNGPallet.Interlock_3,
            Status => "PalletNGData".UnLoadingNGPallet.Status_3,
            Ready => "PalletNGData".UnLoadingNGPallet.Ready_3);
END_REGION

REGION Network 15: InterLock
   RUNG wire#powerrail
      Contact( "AlwaysTRUE" )
      wire#w1
      Contact( "ST10Cylinder".Cy[12].In.WorkPositionSensor )
      I_Contact( "ST10Cylinder".Cy[12].In.HomePositionSensor )
      Coil( "PalletNGData".UnLoadingNGPallet.Interlock_1[1] )
   END_RUNG
   RUNG wire#w1
      Contact( "iE-NG-02Detection" )
      Coil( "PalletNGData".UnLoadingNGPallet.Interlock_1[2] )
   END_RUNG
   RUNG wire#w1
      Coil( "PalletNGData".UnLoadingNGPallet.Interlock_1[3] )
   END_RUNG
   RUNG wire#w1
      Coil( "PalletNGData".UnLoadingNGPallet.Interlock_1[4] )
   END_RUNG
   RUNG wire#w1
      Contact( "PalletNGData".UnLoadingNGPallet.Interlock_1[1] )
      Contact( "PalletNGData".UnLoadingNGPallet.Interlock_1[2] )
      Contact( "PalletNGData".UnLoadingNGPallet.Interlock_1[3] )
      Contact( "PalletNGData".UnLoadingNGPallet.Interlock_1[4] )
      Coil( "PalletNGData".UnLoadingNGPallet.Interlock_1[10] )
      Coil( "PalletNGData".UnLoadingNGPallet.Interlock_2[10] )
      Coil( "PalletNGData".UnLoadingNGPallet.Interlock_3[10] )
   END_RUNG
   // the same network as SCL:
   "PalletNGData".UnLoadingNGPallet.Interlock_1[1] := "AlwaysTRUE" AND "ST10Cylinder".Cy[12].In.WorkPositionSensor AND NOT "ST10Cylinder".Cy[12].In.HomePositionSensor;
   "PalletNGData".UnLoadingNGPallet.Interlock_1[2] := "AlwaysTRUE" AND "iE-NG-02Detection";
   "PalletNGData".UnLoadingNGPallet.Interlock_1[3] := "AlwaysTRUE";
   "PalletNGData".UnLoadingNGPallet.Interlock_1[4] := "AlwaysTRUE";
   #_w1 := "AlwaysTRUE" AND "PalletNGData".UnLoadingNGPallet.Interlock_1[1] AND "PalletNGData".UnLoadingNGPallet.Interlock_1[2] AND "PalletNGData".UnLoadingNGPallet.Interlock_1[3] AND "PalletNGData".UnLoadingNGPallet.Interlock_1[4];
   "PalletNGData".UnLoadingNGPallet.Interlock_1[10] := #_w1;
   "PalletNGData".UnLoadingNGPallet.Interlock_2[10] := #_w1;
   "PalletNGData".UnLoadingNGPallet.Interlock_3[10] := #_w1;
END_REGION

REGION Network 16: NG_Button
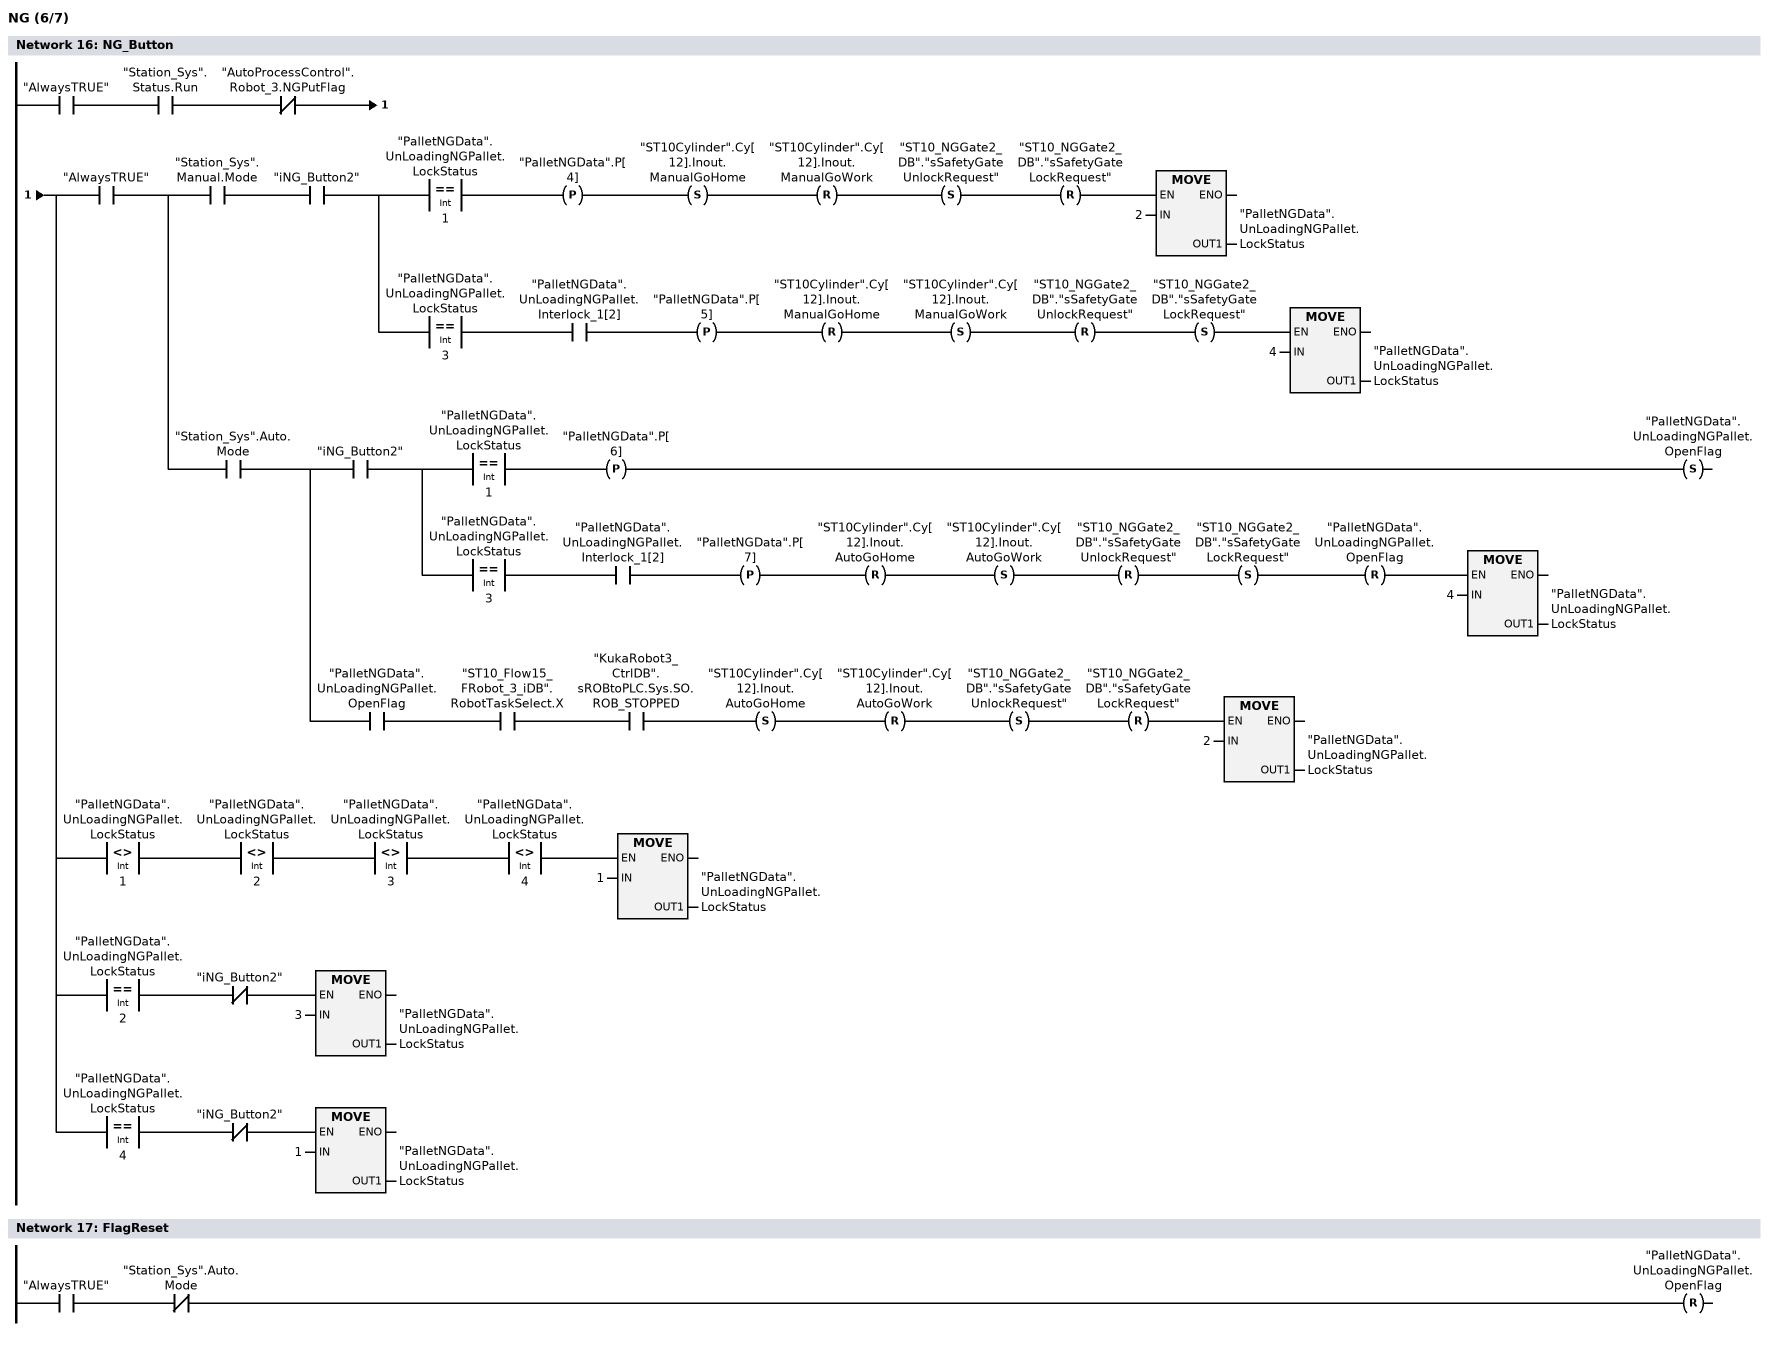
   RUNG wire#powerrail
      Contact( "AlwaysTRUE" )
      Contact( "Station_Sys".Status.Run )
      I_Contact( "AutoProcessControl".Robot_3.NGPutFlag )
      wire#w1
      Contact( "AlwaysTRUE" )
      wire#w2
      Contact( "Station_Sys".Manual.Mode )
      Contact( "iNG_Button2" )
      wire#w3
      { S7_Templates := "SrcType := Int" } EQ_Contact(in1 := "PalletNGData".UnLoadingNGPallet.LockStatus, in2 := 1)
      P_Trig( "PalletNGData".P[4] )
      S_Coil( "ST10Cylinder".Cy[12].Inout.ManualGoHome )
      R_Coil( "ST10Cylinder".Cy[12].Inout.ManualGoWork )
      S_Coil( "ST10_NGGate2_DB"."sSafetyGate UnlockRequest" )
      R_Coil( "ST10_NGGate2_DB"."sSafetyGate LockRequest" )
      Move(in := 2, out1 => "PalletNGData".UnLoadingNGPallet.LockStatus)
   END_RUNG
   RUNG wire#w3
      { S7_Templates := "SrcType := Int" } EQ_Contact(in1 := "PalletNGData".UnLoadingNGPallet.LockStatus, in2 := 3)
      Contact( "PalletNGData".UnLoadingNGPallet.Interlock_1[2] )
      P_Trig( "PalletNGData".P[5] )
      R_Coil( "ST10Cylinder".Cy[12].Inout.ManualGoHome )
      S_Coil( "ST10Cylinder".Cy[12].Inout.ManualGoWork )
      R_Coil( "ST10_NGGate2_DB"."sSafetyGate UnlockRequest" )
      S_Coil( "ST10_NGGate2_DB"."sSafetyGate LockRequest" )
      Move(in := 4, out1 => "PalletNGData".UnLoadingNGPallet.LockStatus)
   END_RUNG
   RUNG wire#w2
      Contact( "Station_Sys".Auto.Mode )
      wire#w4
      Contact( "iNG_Button2" )
      wire#w5
      { S7_Templates := "SrcType := Int" } EQ_Contact(in1 := "PalletNGData".UnLoadingNGPallet.LockStatus, in2 := 1)
      P_Trig( "PalletNGData".P[6] )
      S_Coil( "PalletNGData".UnLoadingNGPallet.OpenFlag )
   END_RUNG
   RUNG wire#w5
      { S7_Templates := "SrcType := Int" } EQ_Contact(in1 := "PalletNGData".UnLoadingNGPallet.LockStatus, in2 := 3)
      Contact( "PalletNGData".UnLoadingNGPallet.Interlock_1[2] )
      P_Trig( "PalletNGData".P[7] )
      R_Coil( "ST10Cylinder".Cy[12].Inout.AutoGoHome )
      S_Coil( "ST10Cylinder".Cy[12].Inout.AutoGoWork )
      R_Coil( "ST10_NGGate2_DB"."sSafetyGate UnlockRequest" )
      S_Coil( "ST10_NGGate2_DB"."sSafetyGate LockRequest" )
      R_Coil( "PalletNGData".UnLoadingNGPallet.OpenFlag )
      Move(in := 4, out1 => "PalletNGData".UnLoadingNGPallet.LockStatus)
   END_RUNG
   RUNG wire#w4
      Contact( "PalletNGData".UnLoadingNGPallet.OpenFlag )
      Contact( "ST10_Flow15_FRobot_3_iDB".RobotTaskSelect.X )
      Contact( "KukaRobot3_CtrlDB".sROBtoPLC.Sys.SO.ROB_STOPPED )
      S_Coil( "ST10Cylinder".Cy[12].Inout.AutoGoHome )
      R_Coil( "ST10Cylinder".Cy[12].Inout.AutoGoWork )
      S_Coil( "ST10_NGGate2_DB"."sSafetyGate UnlockRequest" )
      R_Coil( "ST10_NGGate2_DB"."sSafetyGate LockRequest" )
      Move(in := 2, out1 => "PalletNGData".UnLoadingNGPallet.LockStatus)
   END_RUNG
   RUNG wire#w1
      { S7_Templates := "SrcType := Int" } NE_Contact(in1 := "PalletNGData".UnLoadingNGPallet.LockStatus, in2 := 1)
      { S7_Templates := "SrcType := Int" } NE_Contact(in1 := "PalletNGData".UnLoadingNGPallet.LockStatus, in2 := 2)
      { S7_Templates := "SrcType := Int" } NE_Contact(in1 := "PalletNGData".UnLoadingNGPallet.LockStatus, in2 := 3)
      { S7_Templates := "SrcType := Int" } NE_Contact(in1 := "PalletNGData".UnLoadingNGPallet.LockStatus, in2 := 4)
      Move(in := 1, out1 => "PalletNGData".UnLoadingNGPallet.LockStatus)
   END_RUNG
   RUNG wire#w1
      { S7_Templates := "SrcType := Int" } EQ_Contact(in1 := "PalletNGData".UnLoadingNGPallet.LockStatus, in2 := 2)
      I_Contact( "iNG_Button2" )
      Move(in := 3, out1 => "PalletNGData".UnLoadingNGPallet.LockStatus)
   END_RUNG
   RUNG wire#w1
      { S7_Templates := "SrcType := Int" } EQ_Contact(in1 := "PalletNGData".UnLoadingNGPallet.LockStatus, in2 := 4)
      I_Contact( "iNG_Button2" )
      Move(in := 1, out1 => "PalletNGData".UnLoadingNGPallet.LockStatus)
   END_RUNG
   // the same network as SCL:
   #_w1 := "AlwaysTRUE" AND "Station_Sys".Status.Run AND NOT "AutoProcessControl".Robot_3.NGPutFlag;
   #_w2 := #_w1 AND "AlwaysTRUE";
   #_w3 := #_w2 AND "Station_Sys".Manual.Mode AND "iNG_Button2";
   #_w4 := #_w3 AND ("PalletNGData".UnLoadingNGPallet.LockStatus = 1);
   #_w5 := #_w4 AND NOT "PalletNGData".P[4];   // rising edge
   "PalletNGData".P[4] := #_w4;
   IF #_w5 THEN
       "ST10Cylinder".Cy[12].Inout.ManualGoHome := TRUE;
       "ST10Cylinder".Cy[12].Inout.ManualGoWork := FALSE;
       "ST10_NGGate2_DB"."sSafetyGate UnlockRequest" := TRUE;
       "ST10_NGGate2_DB"."sSafetyGate LockRequest" := FALSE;
       "PalletNGData".UnLoadingNGPallet.LockStatus := 2;
   END_IF;
   #_w6 := #_w3 AND ("PalletNGData".UnLoadingNGPallet.LockStatus = 3) AND "PalletNGData".UnLoadingNGPallet.Interlock_1[2];
   #_w7 := #_w6 AND NOT "PalletNGData".P[5];   // rising edge
   "PalletNGData".P[5] := #_w6;
   IF #_w7 THEN
       "ST10Cylinder".Cy[12].Inout.ManualGoHome := FALSE;
       "ST10Cylinder".Cy[12].Inout.ManualGoWork := TRUE;
       "ST10_NGGate2_DB"."sSafetyGate UnlockRequest" := FALSE;
       "ST10_NGGate2_DB"."sSafetyGate LockRequest" := TRUE;
       "PalletNGData".UnLoadingNGPallet.LockStatus := 4;
   END_IF;
   #_w8 := #_w2 AND "Station_Sys".Auto.Mode;
   #_w9 := #_w8 AND "iNG_Button2";
   #_w10 := #_w9 AND ("PalletNGData".UnLoadingNGPallet.LockStatus = 1);
   #_w11 := #_w10 AND NOT "PalletNGData".P[6];   // rising edge
   "PalletNGData".P[6] := #_w10;
   IF #_w11 THEN "PalletNGData".UnLoadingNGPallet.OpenFlag := TRUE; END_IF;
   #_w12 := #_w9 AND ("PalletNGData".UnLoadingNGPallet.LockStatus = 3) AND "PalletNGData".UnLoadingNGPallet.Interlock_1[2];
   #_w13 := #_w12 AND NOT "PalletNGData".P[7];   // rising edge
   "PalletNGData".P[7] := #_w12;
   IF #_w13 THEN
       "ST10Cylinder".Cy[12].Inout.AutoGoHome := FALSE;
       "ST10Cylinder".Cy[12].Inout.AutoGoWork := TRUE;
       "ST10_NGGate2_DB"."sSafetyGate UnlockRequest" := FALSE;
       "ST10_NGGate2_DB"."sSafetyGate LockRequest" := TRUE;
       "PalletNGData".UnLoadingNGPallet.OpenFlag := FALSE;
       "PalletNGData".UnLoadingNGPallet.LockStatus := 4;
   END_IF;
   IF #_w8 AND "PalletNGData".UnLoadingNGPallet.OpenFlag AND "ST10_Flow15_FRobot_3_iDB".RobotTaskSelect.X AND "KukaRobot3_CtrlDB".sROBtoPLC.Sys.SO.ROB_STOPPED THEN
       "ST10Cylinder".Cy[12].Inout.AutoGoHome := TRUE;
       "ST10Cylinder".Cy[12].Inout.AutoGoWork := FALSE;
       "ST10_NGGate2_DB"."sSafetyGate UnlockRequest" := TRUE;
       "ST10_NGGate2_DB"."sSafetyGate LockRequest" := FALSE;
       "PalletNGData".UnLoadingNGPallet.LockStatus := 2;
   END_IF;
   IF #_w1 AND ("PalletNGData".UnLoadingNGPallet.LockStatus <> 1) AND ("PalletNGData".UnLoadingNGPallet.LockStatus <> 2) AND ("PalletNGData".UnLoadingNGPallet.LockStatus <> 3) AND ("PalletNGData".UnLoadingNGPallet.LockStatus <> 4) THEN
       "PalletNGData".UnLoadingNGPallet.LockStatus := 1;
   END_IF;
   IF #_w1 AND ("PalletNGData".UnLoadingNGPallet.LockStatus = 2) AND NOT "iNG_Button2" THEN
       "PalletNGData".UnLoadingNGPallet.LockStatus := 3;
   END_IF;
   IF #_w1 AND ("PalletNGData".UnLoadingNGPallet.LockStatus = 4) AND NOT "iNG_Button2" THEN
       "PalletNGData".UnLoadingNGPallet.LockStatus := 1;
   END_IF;
END_REGION

REGION Network 17: FlagReset
   RUNG wire#powerrail
      Contact( "AlwaysTRUE" )
      I_Contact( "Station_Sys".Auto.Mode )
      R_Coil( "PalletNGData".UnLoadingNGPallet.OpenFlag )
   END_RUNG
   // the same network as SCL:
   IF "AlwaysTRUE" AND NOT "Station_Sys".Auto.Mode THEN
       "PalletNGData".UnLoadingNGPallet.OpenFlag := FALSE;
   END_IF;
END_REGION

REGION Network 18: NG Door
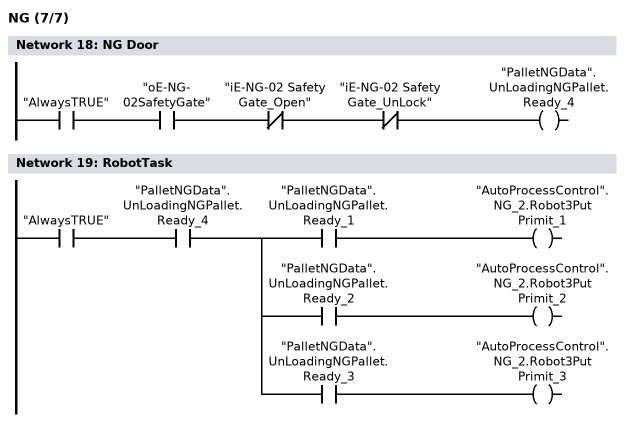
   RUNG wire#powerrail
      Contact( "AlwaysTRUE" )
      Contact( "oE-NG-02SafetyGate" )
      I_Contact( "iE-NG-02 Safety Gate_Open" )
      I_Contact( "iE-NG-02 Safety Gate_UnLock" )
      Coil( "PalletNGData".UnLoadingNGPallet.Ready_4 )
   END_RUNG
   // the same network as SCL:
   "PalletNGData".UnLoadingNGPallet.Ready_4 := "AlwaysTRUE" AND "oE-NG-02SafetyGate" AND NOT "iE-NG-02 Safety Gate_Open" AND NOT "iE-NG-02 Safety Gate_UnLock";
END_REGION

REGION Network 19: RobotTask
   RUNG wire#powerrail
      Contact( "AlwaysTRUE" )
      Contact( "PalletNGData".UnLoadingNGPallet.Ready_4 )
      wire#w1
      Contact( "PalletNGData".UnLoadingNGPallet.Ready_1 )
      Coil( "AutoProcessControl".NG_2.Robot3PutPrimit_1 )
   END_RUNG
   RUNG wire#w1
      Contact( "PalletNGData".UnLoadingNGPallet.Ready_2 )
      Coil( "AutoProcessControl".NG_2.Robot3PutPrimit_2 )
   END_RUNG
   RUNG wire#w1
      Contact( "PalletNGData".UnLoadingNGPallet.Ready_3 )
      Coil( "AutoProcessControl".NG_2.Robot3PutPrimit_3 )
   END_RUNG
   // the same network as SCL:
   #_w1 := "AlwaysTRUE" AND "PalletNGData".UnLoadingNGPallet.Ready_4;
   "AutoProcessControl".NG_2.Robot3PutPrimit_1 := #_w1 AND "PalletNGData".UnLoadingNGPallet.Ready_1;
   "AutoProcessControl".NG_2.Robot3PutPrimit_2 := #_w1 AND "PalletNGData".UnLoadingNGPallet.Ready_2;
   "AutoProcessControl".NG_2.Robot3PutPrimit_3 := #_w1 AND "PalletNGData".UnLoadingNGPallet.Ready_3;
END_REGION
END_FUNCTION_BLOCK

FUNCTION_BLOCK "NGStatus"   // FB2900, LAD
{ S7_Optimized_Access := 'TRUE' }
// stored: AutoNumber false, MemoryReserve 100, SetENOAutomatically false
   VAR_INPUT
      NG_1 : Bool;
      NG_2 : Bool;
      NG_3 : Bool;
      NG_4 : Bool;
      NG_5 : Bool;
   END_VAR
   VAR_OUTPUT
      Status : Int;
      Ready : Bool;
   END_VAR
   VAR_IN_OUT
      Interlock : Array[1..10] of Bool;
   END_VAR
   VAR
      AlwaysOn : Bool;
      NG_Delay : Array[1..10] of TON_TIME;
      NG_DelayTime { S7_SetPoint := 'True'} : Array[1..10] of DInt;
   END_VAR
   // NG_DelayTime[1..10] := 1000;
BEGIN

REGION Network 1: #AlwaysOn
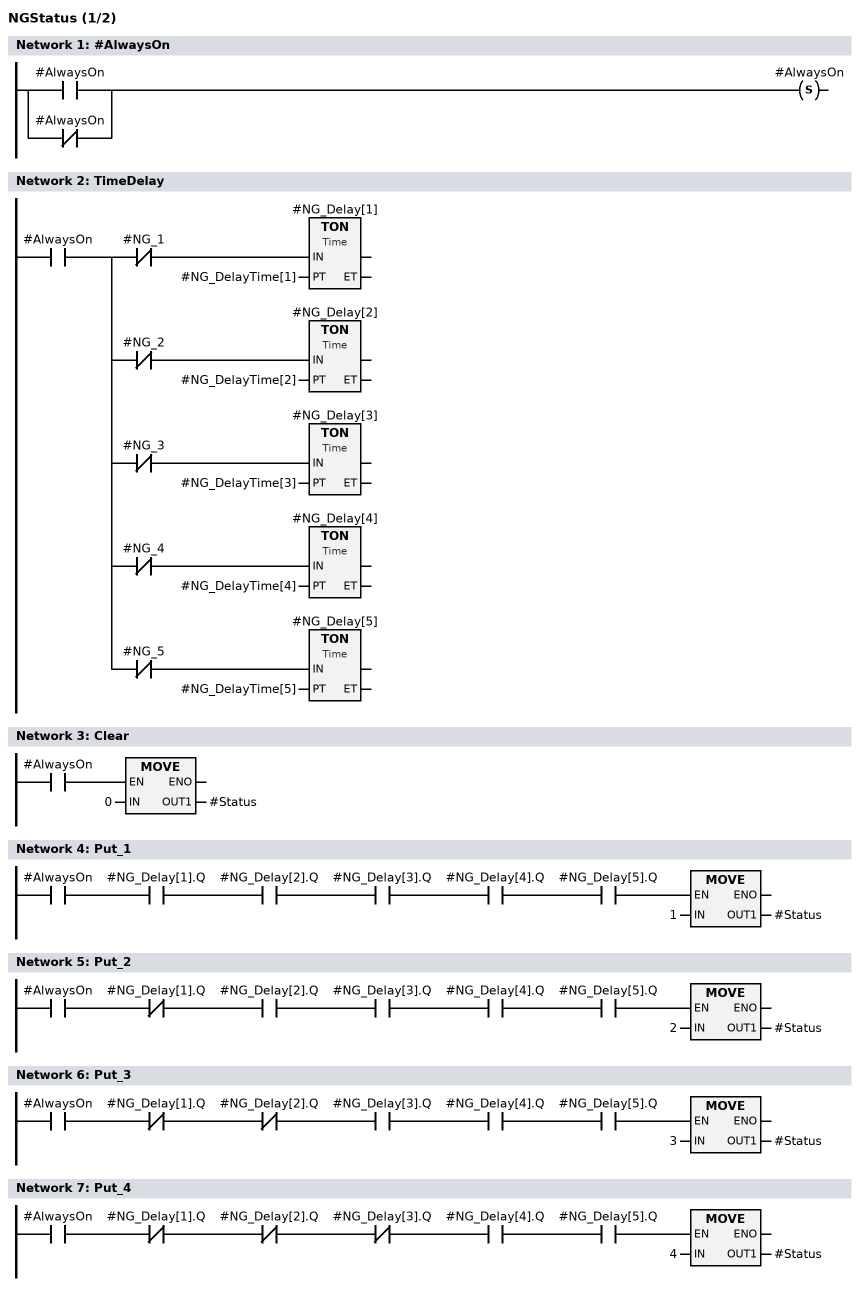
   RUNG wire#powerrail
      Contact( #AlwaysOn )
      wire#w1
      S_Coil( #AlwaysOn )
   END_RUNG
   RUNG wire#powerrail
      I_Contact( #AlwaysOn )
   END_RUNG wire#w1
   // the same network as SCL:
   IF #AlwaysOn OR NOT #AlwaysOn THEN #AlwaysOn := TRUE; END_IF;
END_REGION

REGION Network 2: TimeDelay
   RUNG wire#powerrail
      Contact( #AlwaysOn )
      wire#w1
      I_Contact( #NG_1 )
      { S7_Templates := "time_type := Time" } #NG_Delay[1].TON(pt := #NG_DelayTime[1], et =>)
   END_RUNG
   RUNG wire#w1
      I_Contact( #NG_2 )
      { S7_Templates := "time_type := Time" } #NG_Delay[2].TON(pt := #NG_DelayTime[2], et =>)
   END_RUNG
   RUNG wire#w1
      I_Contact( #NG_3 )
      { S7_Templates := "time_type := Time" } #NG_Delay[3].TON(pt := #NG_DelayTime[3], et =>)
   END_RUNG
   RUNG wire#w1
      I_Contact( #NG_4 )
      { S7_Templates := "time_type := Time" } #NG_Delay[4].TON(pt := #NG_DelayTime[4], et =>)
   END_RUNG
   RUNG wire#w1
      I_Contact( #NG_5 )
      { S7_Templates := "time_type := Time" } #NG_Delay[5].TON(pt := #NG_DelayTime[5], et =>)
   END_RUNG
   // the same network as SCL:
   #NG_Delay[1].TON(IN := #AlwaysOn AND NOT #NG_1, PT := #NG_DelayTime[1]);
   #NG_Delay[2].TON(IN := #AlwaysOn AND NOT #NG_2, PT := #NG_DelayTime[2]);
   #NG_Delay[3].TON(IN := #AlwaysOn AND NOT #NG_3, PT := #NG_DelayTime[3]);
   #NG_Delay[4].TON(IN := #AlwaysOn AND NOT #NG_4, PT := #NG_DelayTime[4]);
   #NG_Delay[5].TON(IN := #AlwaysOn AND NOT #NG_5, PT := #NG_DelayTime[5]);
END_REGION

REGION Network 3: Clear
   RUNG wire#powerrail
      Contact( #AlwaysOn )
      Move(in := 0, out1 => #Status)
   END_RUNG
   // the same network as SCL:
   IF #AlwaysOn THEN #Status := 0; END_IF;
END_REGION

REGION Network 4: Put_1
   RUNG wire#powerrail
      Contact( #AlwaysOn )
      Contact( #NG_Delay[1].Q )
      Contact( #NG_Delay[2].Q )
      Contact( #NG_Delay[3].Q )
      Contact( #NG_Delay[4].Q )
      Contact( #NG_Delay[5].Q )
      Move(in := 1, out1 => #Status)
   END_RUNG
   // the same network as SCL:
   IF #AlwaysOn AND #NG_Delay[1].Q AND #NG_Delay[2].Q AND #NG_Delay[3].Q AND #NG_Delay[4].Q AND #NG_Delay[5].Q THEN
       #Status := 1;
   END_IF;
END_REGION

REGION Network 5: Put_2
   RUNG wire#powerrail
      Contact( #AlwaysOn )
      I_Contact( #NG_Delay[1].Q )
      Contact( #NG_Delay[2].Q )
      Contact( #NG_Delay[3].Q )
      Contact( #NG_Delay[4].Q )
      Contact( #NG_Delay[5].Q )
      Move(in := 2, out1 => #Status)
   END_RUNG
   // the same network as SCL:
   IF #AlwaysOn AND NOT #NG_Delay[1].Q AND #NG_Delay[2].Q AND #NG_Delay[3].Q AND #NG_Delay[4].Q AND #NG_Delay[5].Q THEN
       #Status := 2;
   END_IF;
END_REGION

REGION Network 6: Put_3
   RUNG wire#powerrail
      Contact( #AlwaysOn )
      I_Contact( #NG_Delay[1].Q )
      I_Contact( #NG_Delay[2].Q )
      Contact( #NG_Delay[3].Q )
      Contact( #NG_Delay[4].Q )
      Contact( #NG_Delay[5].Q )
      Move(in := 3, out1 => #Status)
   END_RUNG
   // the same network as SCL:
   IF #AlwaysOn AND NOT #NG_Delay[1].Q AND NOT #NG_Delay[2].Q AND #NG_Delay[3].Q AND #NG_Delay[4].Q AND #NG_Delay[5].Q THEN
       #Status := 3;
   END_IF;
END_REGION

REGION Network 7: Put_4
   RUNG wire#powerrail
      Contact( #AlwaysOn )
      I_Contact( #NG_Delay[1].Q )
      I_Contact( #NG_Delay[2].Q )
      I_Contact( #NG_Delay[3].Q )
      Contact( #NG_Delay[4].Q )
      Contact( #NG_Delay[5].Q )
      Move(in := 4, out1 => #Status)
   END_RUNG
   // the same network as SCL:
   IF #AlwaysOn AND NOT #NG_Delay[1].Q AND NOT #NG_Delay[2].Q AND NOT #NG_Delay[3].Q AND #NG_Delay[4].Q AND #NG_Delay[5].Q THEN
       #Status := 4;
   END_IF;
END_REGION

REGION Network 8: Put_5
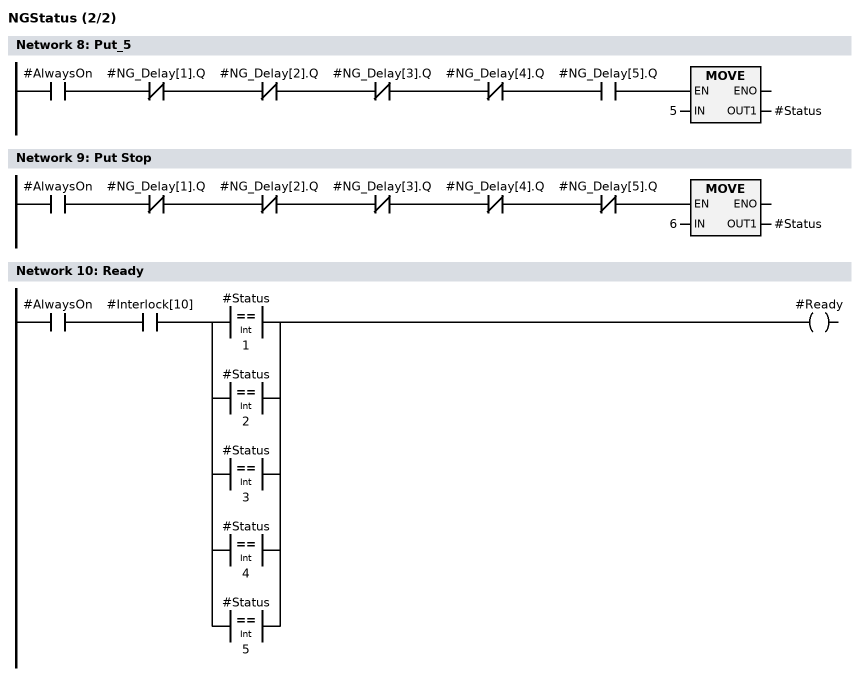
   RUNG wire#powerrail
      Contact( #AlwaysOn )
      I_Contact( #NG_Delay[1].Q )
      I_Contact( #NG_Delay[2].Q )
      I_Contact( #NG_Delay[3].Q )
      I_Contact( #NG_Delay[4].Q )
      Contact( #NG_Delay[5].Q )
      Move(in := 5, out1 => #Status)
   END_RUNG
   // the same network as SCL:
   IF #AlwaysOn AND NOT #NG_Delay[1].Q AND NOT #NG_Delay[2].Q AND NOT #NG_Delay[3].Q AND NOT #NG_Delay[4].Q AND #NG_Delay[5].Q THEN
       #Status := 5;
   END_IF;
END_REGION

REGION Network 9: Put Stop
   RUNG wire#powerrail
      Contact( #AlwaysOn )
      I_Contact( #NG_Delay[1].Q )
      I_Contact( #NG_Delay[2].Q )
      I_Contact( #NG_Delay[3].Q )
      I_Contact( #NG_Delay[4].Q )
      I_Contact( #NG_Delay[5].Q )
      Move(in := 6, out1 => #Status)
   END_RUNG
   // the same network as SCL:
   IF #AlwaysOn AND NOT #NG_Delay[1].Q AND NOT #NG_Delay[2].Q AND NOT #NG_Delay[3].Q AND NOT #NG_Delay[4].Q AND NOT #NG_Delay[5].Q THEN
       #Status := 6;
   END_IF;
END_REGION

REGION Network 10: Ready
   RUNG wire#powerrail
      Contact( #AlwaysOn )
      Contact( #Interlock[10] )
      wire#w1
      { S7_Templates := "SrcType := Int" } EQ_Contact(in1 := #Status, in2 := 1)
      wire#w2
      Coil( #Ready )
   END_RUNG
   RUNG wire#w1
      { S7_Templates := "SrcType := Int" } EQ_Contact(in1 := #Status, in2 := 2)
   END_RUNG wire#w2
   RUNG wire#w1
      { S7_Templates := "SrcType := Int" } EQ_Contact(in1 := #Status, in2 := 3)
   END_RUNG wire#w2
   RUNG wire#w1
      { S7_Templates := "SrcType := Int" } EQ_Contact(in1 := #Status, in2 := 4)
   END_RUNG wire#w2
   RUNG wire#w1
      { S7_Templates := "SrcType := Int" } EQ_Contact(in1 := #Status, in2 := 5)
   END_RUNG wire#w2
   // the same network as SCL:
   #Ready := #AlwaysOn AND #Interlock[10] AND ((#Status = 1) OR (#Status = 2) OR (#Status = 3) OR (#Status = 4) OR (#Status = 5));
END_REGION
END_FUNCTION_BLOCK

FUNCTION "MES" : Void   // FC500, LAD
{ S7_Optimized_Access := 'TRUE' }
// stored: AutoNumber false, SetENOAutomatically false
   VAR_TEMP
      YEAR : Int;
      MONTH : Int;
      DAY : Int;
      HH : Int;
      MM : Int;
      SS : Int;
      RET1 : Int;
      RET2 : Int;
      P : Array[0..10] of Bool;
   END_VAR
   VAR_TEMP   // added for the SCL form of the ladder/FBD networks
      _w1 : Bool;
      _w2 : Bool;
   END_VAR
BEGIN

REGION Network 2: 自动复位测试 / Automatic reset test
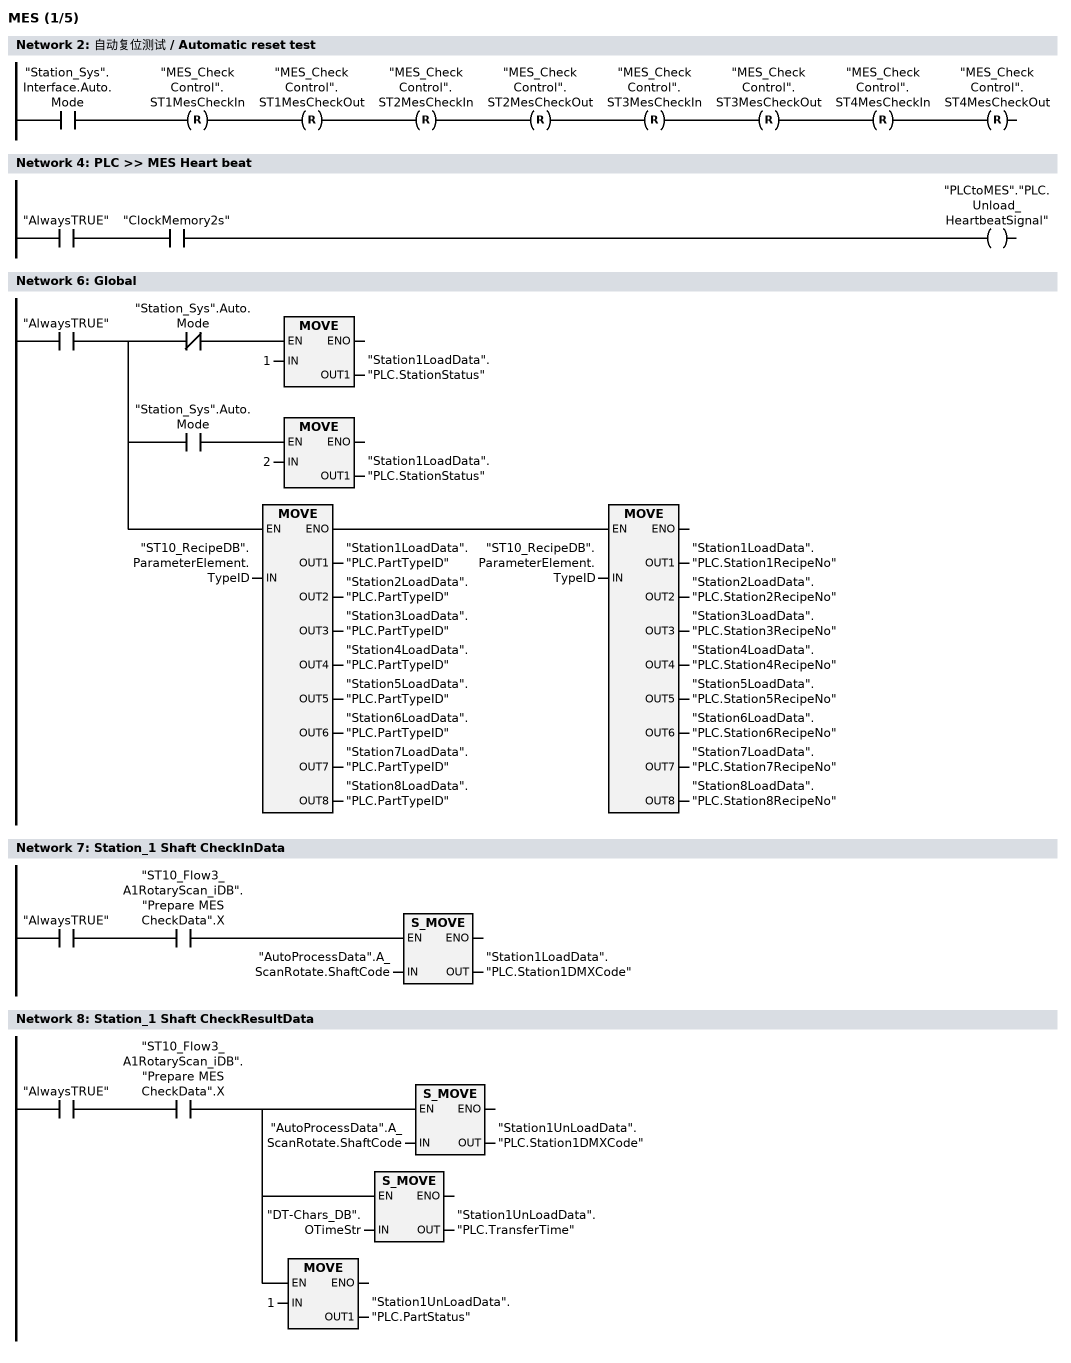
   RUNG wire#powerrail
      Contact( "Station_Sys".Interface.Auto.Mode )
      R_Coil( "MES_CheckControl".ST1MesCheckIn )
      R_Coil( "MES_CheckControl".ST1MesCheckOut )
      R_Coil( "MES_CheckControl".ST2MesCheckIn )
      R_Coil( "MES_CheckControl".ST2MesCheckOut )
      R_Coil( "MES_CheckControl".ST3MesCheckIn )
      R_Coil( "MES_CheckControl".ST3MesCheckOut )
      R_Coil( "MES_CheckControl".ST4MesCheckIn )
      R_Coil( "MES_CheckControl".ST4MesCheckOut )
   END_RUNG
   // the same network as SCL:
   IF "Station_Sys".Interface.Auto.Mode THEN
       "MES_CheckControl".ST1MesCheckIn := FALSE;
       "MES_CheckControl".ST1MesCheckOut := FALSE;
       "MES_CheckControl".ST2MesCheckIn := FALSE;
       "MES_CheckControl".ST2MesCheckOut := FALSE;
       "MES_CheckControl".ST3MesCheckIn := FALSE;
       "MES_CheckControl".ST3MesCheckOut := FALSE;
       "MES_CheckControl".ST4MesCheckIn := FALSE;
       "MES_CheckControl".ST4MesCheckOut := FALSE;
   END_IF;
END_REGION

NETWORK
TITLE = PLC系统时间转换 / PLC system time conversion
//########提取PLC当前日期
      L     %DB3000.DBB18;
      BTI;
      T     #YEAR;
      L     %DB3000.DBB19;
      BTI;
      T     #MONTH;
      L     %DB3000.DBB20;
      BTI;
      T     #DAY;
      L     %DB3000.DBB21;
      BTI;
      T     #HH;
      L     %DB3000.DBB22;
      BTI;
      T     #MM;
      L     %DB3000.DBB23;
      BTI;
      T     #SS;


//########将日期转化成字符
      CALL  "DT-Chars", "DT-Chars_DB"
      ( YEAR                := #YEAR,
        MONTH               := #MONTH,
        DAY                 := #DAY,
        HH                  := #HH,
        MM                  := #MM,
        SS                  := #SS,
        Year_Byte1          := ,
        Year_Byte2          := ,
        Month_Byte1         := ,
        Month_Byte2         := ,
        Days_Byte1          := ,
        Days_Byte2          := ,
        HH_Byte1            := ,
        HH_Byte2            := ,
        MM_Byte1            := ,
        MM_Byte2            := ,
        SS_Byte1            := ,
        SS_Byte2            := ,
        CalculateDays_Byte1 := ,
        CalculateDays_Byte2 := ,
        CalculateDays_Byte3 := ,
        Error_Code          := ,
        Year_Byte3          := ,
        Year_Byte4          := ,
        Month_Byte3         := ,
        Month_Byte4         := ,
        Days_Byte3          := ,
        Days_Byte4          := ,
        HH_Byte3            := ,
        HH_Byte4            := ,
        MM_Byte3            := ,
        MM_Byte4            := ,
        SS_Byte3            := ,
        SS_Byte4            := ,
        CalculateDays_Byte4 := ,
        CalculateDays_Byte5 := ,
        CalculateDays_Byte6 := ,
        OTimeStr            := 
      );




REGION Network 4: PLC >> MES Heart beat
   RUNG wire#powerrail
      Contact( "AlwaysTRUE" )
      Contact( "ClockMemory2s" )
      Coil( "PLCtoMES"."PLC.Unload_HeartbeatSignal" )
   END_RUNG
   // the same network as SCL:
   "PLCtoMES"."PLC.Unload_HeartbeatSignal" := "AlwaysTRUE" AND "ClockMemory2s";
END_REGION

REGION Network 6: Global
   RUNG wire#powerrail
      Contact( "AlwaysTRUE" )
      wire#w1
      I_Contact( "Station_Sys".Auto.Mode )
      Move(in := 1, out1 => "Station1LoadData"."PLC.StationStatus")
   END_RUNG
   RUNG wire#w1
      Contact( "Station_Sys".Auto.Mode )
      Move(in := 2, out1 => "Station1LoadData"."PLC.StationStatus")
   END_RUNG
   RUNG wire#w1
      Move(in := "ST10_RecipeDB".ParameterElement.TypeID, out1 => "Station1LoadData"."PLC.PartTypeID", out2 => "Station2LoadData"."PLC.PartTypeID", out3 => "Station3LoadData"."PLC.PartTypeID", out4 => "Station4LoadData"."PLC.PartTypeID", out5 => "Station5LoadData"."PLC.PartTypeID", out6 => "Station6LoadData"."PLC.PartTypeID", out7 => "Station7LoadData"."PLC.PartTypeID", out8 => "Station8LoadData"."PLC.PartTypeID")
      Move(in := "ST10_RecipeDB".ParameterElement.TypeID, out1 => "Station1LoadData"."PLC.Station1RecipeNo", out2 => "Station2LoadData"."PLC.Station2RecipeNo", out3 => "Station3LoadData"."PLC.Station3RecipeNo", out4 => "Station4LoadData"."PLC.Station4RecipeNo", out5 => "Station5LoadData"."PLC.Station5RecipeNo", out6 => "Station6LoadData"."PLC.Station6RecipeNo", out7 => "Station7LoadData"."PLC.Station7RecipeNo", out8 => "Station8LoadData"."PLC.Station8RecipeNo")
   END_RUNG
   // the same network as SCL:
   IF "AlwaysTRUE" AND NOT "Station_Sys".Auto.Mode THEN "Station1LoadData"."PLC.StationStatus" := 1; END_IF;
   IF "AlwaysTRUE" AND "Station_Sys".Auto.Mode THEN "Station1LoadData"."PLC.StationStatus" := 2; END_IF;
   IF "AlwaysTRUE" THEN
       "Station1LoadData"."PLC.PartTypeID" := "ST10_RecipeDB".ParameterElement.TypeID;
       "Station2LoadData"."PLC.PartTypeID" := "ST10_RecipeDB".ParameterElement.TypeID;
       "Station3LoadData"."PLC.PartTypeID" := "ST10_RecipeDB".ParameterElement.TypeID;
       "Station4LoadData"."PLC.PartTypeID" := "ST10_RecipeDB".ParameterElement.TypeID;
       "Station5LoadData"."PLC.PartTypeID" := "ST10_RecipeDB".ParameterElement.TypeID;
       "Station6LoadData"."PLC.PartTypeID" := "ST10_RecipeDB".ParameterElement.TypeID;
       "Station7LoadData"."PLC.PartTypeID" := "ST10_RecipeDB".ParameterElement.TypeID;
       "Station8LoadData"."PLC.PartTypeID" := "ST10_RecipeDB".ParameterElement.TypeID;
       "Station1LoadData"."PLC.Station1RecipeNo" := "ST10_RecipeDB".ParameterElement.TypeID;
       "Station2LoadData"."PLC.Station2RecipeNo" := "ST10_RecipeDB".ParameterElement.TypeID;
       "Station3LoadData"."PLC.Station3RecipeNo" := "ST10_RecipeDB".ParameterElement.TypeID;
       "Station4LoadData"."PLC.Station4RecipeNo" := "ST10_RecipeDB".ParameterElement.TypeID;
       "Station5LoadData"."PLC.Station5RecipeNo" := "ST10_RecipeDB".ParameterElement.TypeID;
       "Station6LoadData"."PLC.Station6RecipeNo" := "ST10_RecipeDB".ParameterElement.TypeID;
       "Station7LoadData"."PLC.Station7RecipeNo" := "ST10_RecipeDB".ParameterElement.TypeID;
       "Station8LoadData"."PLC.Station8RecipeNo" := "ST10_RecipeDB".ParameterElement.TypeID;
   END_IF;
END_REGION

